  PROC DrawPart165()
    MoveL Offs(pOrigin,280.39,171.29,0.00),v40,z0,tPen\WObj:=wPaper;
    MoveL Offs(pOrigin,280.60,172.34,0.00),v40,z0,tPen\WObj:=wPaper;
    MoveL Offs(pOrigin,279.54,172.34,0.00),v40,fine,tPen\WObj:=wPaper;
    MoveL Offs(pOrigin,279.54,172.34,6.00),v60,z5,tPen\WObj:=wPaper;
    MoveL Offs(pOrigin,278.38,172.88,6.00),vTravel,z5,tPen\WObj:=wPaper;
    MoveL Offs(pOrigin,278.38,172.88,0.00),v60,z0,tPen\WObj:=wPaper;
    MoveL Offs(pOrigin,281.24,170.02,0.00),v40,fine,tPen\WObj:=wPaper;
    MoveL Offs(pOrigin,281.24,170.02,6.00),v60,z5,tPen\WObj:=wPaper;
    MoveL Offs(pOrigin,281.53,171.22,6.00),vTravel,z5,tPen\WObj:=wPaper;
    MoveL Offs(pOrigin,281.53,171.22,0.00),v60,z0,tPen\WObj:=wPaper;
    MoveL Offs(pOrigin,278.68,174.08,0.00),v40,fine,tPen\WObj:=wPaper;
    MoveL Offs(pOrigin,278.68,174.08,6.00),v60,z5,tPen\WObj:=wPaper;
    MoveL Offs(pOrigin,279.85,175.00,6.00),vTravel,z5,tPen\WObj:=wPaper;
    MoveL Offs(pOrigin,279.85,175.00,0.00),v60,z0,tPen\WObj:=wPaper;
    MoveL Offs(pOrigin,279.85,176.91,0.00),v40,z0,tPen\WObj:=wPaper;
    MoveL Offs(pOrigin,280.91,177.12,0.00),v40,z0,tPen\WObj:=wPaper;
    MoveL Offs(pOrigin,280.91,175.42,0.00),v40,z0,tPen\WObj:=wPaper;
    MoveL Offs(pOrigin,281.45,175.51,0.00),v40,z0,tPen\WObj:=wPaper;
    MoveL Offs(pOrigin,279.32,175.51,0.00),v40,z0,tPen\WObj:=wPaper;
    MoveL Offs(pOrigin,278.53,175.77,0.00),v40,z0,tPen\WObj:=wPaper;
    MoveL Offs(pOrigin,283.18,180.43,0.00),v40,z0,tPen\WObj:=wPaper;
    MoveL Offs(pOrigin,283.30,179.90,0.00),v40,z0,tPen\WObj:=wPaper;
    MoveL Offs(pOrigin,280.75,182.46,0.00),v40,z0,tPen\WObj:=wPaper;
    MoveL Offs(pOrigin,281.40,183.12,0.00),v40,z0,tPen\WObj:=wPaper;
    MoveL Offs(pOrigin,284.70,186.43,0.00),v40,z0,tPen\WObj:=wPaper;
    MoveL Offs(pOrigin,284.78,185.89,0.00),v40,z0,tPen\WObj:=wPaper;
    MoveL Offs(pOrigin,282.23,188.45,0.00),v40,z0,tPen\WObj:=wPaper;
    MoveL Offs(pOrigin,282.76,188.97,0.00),v40,z0,tPen\WObj:=wPaper;
    MoveL Offs(pOrigin,286.07,192.28,0.00),v40,z0,tPen\WObj:=wPaper;
    MoveL Offs(pOrigin,286.26,191.88,0.00),v40,z0,tPen\WObj:=wPaper;
    MoveL Offs(pOrigin,283.86,194.28,0.00),v40,z0,tPen\WObj:=wPaper;
    MoveL Offs(pOrigin,284.28,194.97,0.00),v40,z0,tPen\WObj:=wPaper;
    MoveL Offs(pOrigin,288.33,199.02,0.00),v40,z0,tPen\WObj:=wPaper;
    MoveL Offs(pOrigin,287.61,199.80,0.00),v40,z0,tPen\WObj:=wPaper;
    MoveL Offs(pOrigin,286.34,199.80,0.00),v40,z0,tPen\WObj:=wPaper;
    MoveL Offs(pOrigin,286.55,200.86,0.00),v40,z0,tPen\WObj:=wPaper;
    MoveL Offs(pOrigin,287.61,200.86,0.00),v40,z0,tPen\WObj:=wPaper;
    MoveL Offs(pOrigin,288.63,201.46,0.00),v40,z0,tPen\WObj:=wPaper;
    MoveL Offs(pOrigin,286.07,204.01,0.00),v40,z0,tPen\WObj:=wPaper;
    MoveL Offs(pOrigin,287.19,204.02,0.00),v40,z0,tPen\WObj:=wPaper;
    MoveL Offs(pOrigin,288.25,204.02,0.00),v40,z0,tPen\WObj:=wPaper;
    MoveL Offs(pOrigin,288.46,205.08,0.00),v40,z0,tPen\WObj:=wPaper;
    MoveL Offs(pOrigin,287.40,205.08,0.00),v40,fine,tPen\WObj:=wPaper;
    MoveL Offs(pOrigin,287.40,205.08,6.00),v60,z5,tPen\WObj:=wPaper;
    MoveL Offs(pOrigin,289.52,205.05,6.00),vTravel,z5,tPen\WObj:=wPaper;
    MoveL Offs(pOrigin,289.52,205.05,0.00),v60,z0,tPen\WObj:=wPaper;
    MoveL Offs(pOrigin,286.66,207.91,0.00),v40,z0,tPen\WObj:=wPaper;
    MoveL Offs(pOrigin,287.32,208.46,0.00),v40,z0,tPen\WObj:=wPaper;
    MoveL Offs(pOrigin,289.87,211.01,0.00),v40,z0,tPen\WObj:=wPaper;
    MoveL Offs(pOrigin,290.25,210.29,0.00),v40,z0,tPen\WObj:=wPaper;
    MoveL Offs(pOrigin,287.55,213.00,0.00),v40,z0,tPen\WObj:=wPaper;
    MoveL Offs(pOrigin,287.93,213.55,0.00),v40,z0,tPen\WObj:=wPaper;
    MoveL Offs(pOrigin,290.03,215.66,0.00),v40,z0,tPen\WObj:=wPaper;
    MoveL Offs(pOrigin,290.83,215.68,0.00),v40,z0,tPen\WObj:=wPaper;
    MoveL Offs(pOrigin,284.07,222.44,0.00),v40,z0,tPen\WObj:=wPaper;
    MoveL Offs(pOrigin,284.82,223.19,0.00),v40,z0,tPen\WObj:=wPaper;
    MoveL Offs(pOrigin,290.83,217.18,0.00),v40,z0,tPen\WObj:=wPaper;
    MoveL Offs(pOrigin,290.04,217.15,0.00),v40,z0,tPen\WObj:=wPaper;
    MoveL Offs(pOrigin,288.08,215.20,0.00),v40,z0,tPen\WObj:=wPaper;
    MoveL Offs(pOrigin,287.54,214.49,0.00),v40,z0,tPen\WObj:=wPaper;
    MoveL Offs(pOrigin,290.40,211.64,0.00),v40,z0,tPen\WObj:=wPaper;
    MoveL Offs(pOrigin,289.87,212.51,0.00),v40,z0,tPen\WObj:=wPaper;
    MoveL Offs(pOrigin,287.77,210.41,0.00),v40,z0,tPen\WObj:=wPaper;
    MoveL Offs(pOrigin,288.25,210.36,0.00),v40,z0,tPen\WObj:=wPaper;
    MoveL Offs(pOrigin,289.31,210.36,0.00),v40,fine,tPen\WObj:=wPaper;
    MoveL Offs(pOrigin,289.31,210.36,6.00),v60,z5,tPen\WObj:=wPaper;
    MoveL Offs(pOrigin,287.10,210.45,6.00),vTravel,z5,tPen\WObj:=wPaper;
    MoveL Offs(pOrigin,287.10,210.45,0.00),v60,z0,tPen\WObj:=wPaper;
    MoveL Offs(pOrigin,289.96,207.60,0.00),v40,fine,tPen\WObj:=wPaper;
    MoveL Offs(pOrigin,289.96,207.60,6.00),v60,z5,tPen\WObj:=wPaper;
    MoveL Offs(pOrigin,289.81,206.25,6.00),vTravel,z5,tPen\WObj:=wPaper;
    MoveL Offs(pOrigin,289.81,206.25,0.00),v60,z0,tPen\WObj:=wPaper;
    MoveL Offs(pOrigin,286.96,209.10,0.00),v40,fine,tPen\WObj:=wPaper;
    MoveL Offs(pOrigin,286.96,209.10,6.00),v60,z5,tPen\WObj:=wPaper;
    MoveL Offs(pOrigin,284.26,210.31,6.00),vTravel,z5,tPen\WObj:=wPaper;
    MoveL Offs(pOrigin,284.26,210.31,0.00),v60,z0,tPen\WObj:=wPaper;
    MoveL Offs(pOrigin,282.00,212.56,0.00),v40,z0,tPen\WObj:=wPaper;
    MoveL Offs(pOrigin,282.23,212.34,0.00),v40,z0,tPen\WObj:=wPaper;
    MoveL Offs(pOrigin,286.74,216.84,0.00),v40,fine,tPen\WObj:=wPaper;
    MoveL Offs(pOrigin,286.74,216.84,6.00),v60,z5,tPen\WObj:=wPaper;
    MoveL Offs(pOrigin,288.09,216.70,6.00),vTravel,z5,tPen\WObj:=wPaper;
    MoveL Offs(pOrigin,288.09,216.70,0.00),v60,z0,tPen\WObj:=wPaper;
    MoveL Offs(pOrigin,290.04,218.65,0.00),v40,z0,tPen\WObj:=wPaper;
    MoveL Offs(pOrigin,290.52,218.98,0.00),v40,z0,tPen\WObj:=wPaper;
    MoveL Offs(pOrigin,285.26,224.24,0.00),v40,z0,tPen\WObj:=wPaper;
    MoveL Offs(pOrigin,285.86,225.13,0.00),v40,z0,tPen\WObj:=wPaper;
    MoveL Offs(pOrigin,290.82,220.18,0.00),v40,z0,tPen\WObj:=wPaper;
    MoveL Offs(pOrigin,291.85,220.46,0.00),v40,z0,tPen\WObj:=wPaper;
    MoveL Offs(pOrigin,293.35,221.96,0.00),v40,z0,tPen\WObj:=wPaper;
    MoveL Offs(pOrigin,292.71,222.18,0.00),v40,z0,tPen\WObj:=wPaper;
    MoveL Offs(pOrigin,292.50,222.60,0.00),v40,z0,tPen\WObj:=wPaper;
    MoveL Offs(pOrigin,292.71,222.18,0.00),v40,z0,tPen\WObj:=wPaper;
    MoveL Offs(pOrigin,292.50,221.98,0.00),v40,z0,tPen\WObj:=wPaper;
    MoveL Offs(pOrigin,291.23,221.98,0.00),v40,z0,tPen\WObj:=wPaper;
    MoveL Offs(pOrigin,291.25,221.35,0.00),v40,z0,tPen\WObj:=wPaper;
    MoveL Offs(pOrigin,292.60,222.70,0.00),v40,z0,tPen\WObj:=wPaper;
    MoveL Offs(pOrigin,292.08,222.81,0.00),v40,z0,tPen\WObj:=wPaper;
    MoveL Offs(pOrigin,291.86,223.24,0.00),v40,z0,tPen\WObj:=wPaper;
    MoveL Offs(pOrigin,292.08,222.81,0.00),v40,z0,tPen\WObj:=wPaper;
    MoveL Offs(pOrigin,291.65,223.03,0.00),v40,z0,tPen\WObj:=wPaper;
    MoveL Offs(pOrigin,286.12,223.03,0.00),v40,z0,tPen\WObj:=wPaper;
    MoveL Offs(pOrigin,286.55,222.39,0.00),v40,z0,tPen\WObj:=wPaper;
    MoveL Offs(pOrigin,286.98,223.66,0.00),v40,z0,tPen\WObj:=wPaper;
    MoveL Offs(pOrigin,286.55,223.88,0.00),v40,z0,tPen\WObj:=wPaper;
    MoveL Offs(pOrigin,286.55,223.88,0.00),v40,z0,tPen\WObj:=wPaper;
    MoveL Offs(pOrigin,285.91,223.45,0.00),v40,z0,tPen\WObj:=wPaper;
    MoveL Offs(pOrigin,283.43,219.62,0.00),v40,z0,tPen\WObj:=wPaper;
    MoveL Offs(pOrigin,283.79,219.48,0.00),v40,z0,tPen\WObj:=wPaper;
    MoveL Offs(pOrigin,284.42,219.84,0.00),v40,z0,tPen\WObj:=wPaper;
    MoveL Offs(pOrigin,285.91,221.96,0.00),v40,z0,tPen\WObj:=wPaper;
    MoveL Offs(pOrigin,286.55,222.39,0.00),v40,z0,tPen\WObj:=wPaper;
    MoveL Offs(pOrigin,286.55,222.39,0.00),v40,z0,tPen\WObj:=wPaper;
    MoveL Offs(pOrigin,286.76,221.54,0.00),v40,z0,tPen\WObj:=wPaper;
    MoveL Offs(pOrigin,284.71,216.01,0.00),v40,z0,tPen\WObj:=wPaper;
    MoveL Offs(pOrigin,282.65,211.76,0.00),v40,z0,tPen\WObj:=wPaper;
    MoveL Offs(pOrigin,279.47,207.30,0.00),v40,z0,tPen\WObj:=wPaper;
    MoveL Offs(pOrigin,278.69,205.39,0.00),v40,z0,tPen\WObj:=wPaper;
    MoveL Offs(pOrigin,272.10,200.64,0.00),v40,z0,tPen\WObj:=wPaper;
    MoveL Offs(pOrigin,267.64,198.38,0.00),v40,fine,tPen\WObj:=wPaper;
    MoveL Offs(pOrigin,267.64,198.38,6.00),v60,z5,tPen\WObj:=wPaper;
  ENDPROC

  PROC DrawPart166()
    MoveL Offs(pOrigin,269.31,199.87,6.00),vTravel,z5,tPen\WObj:=wPaper;
    MoveL Offs(pOrigin,269.31,199.87,0.00),v60,z0,tPen\WObj:=wPaper;
    MoveL Offs(pOrigin,270.51,198.67,0.00),v40,z0,tPen\WObj:=wPaper;
    MoveL Offs(pOrigin,271.56,199.11,0.00),v40,z0,tPen\WObj:=wPaper;
    MoveL Offs(pOrigin,270.21,200.47,0.00),v40,z0,tPen\WObj:=wPaper;
    MoveL Offs(pOrigin,271.10,201.06,0.00),v40,z0,tPen\WObj:=wPaper;
    MoveL Offs(pOrigin,272.46,199.71,0.00),v40,z0,tPen\WObj:=wPaper;
    MoveL Offs(pOrigin,271.86,200.47,0.00),v40,z0,tPen\WObj:=wPaper;
    MoveL Offs(pOrigin,275.62,204.23,0.00),v40,z0,tPen\WObj:=wPaper;
    MoveL Offs(pOrigin,275.14,204.50,0.00),v40,z0,tPen\WObj:=wPaper;
    MoveL Offs(pOrigin,279.04,200.59,0.00),v40,z0,tPen\WObj:=wPaper;
    MoveL Offs(pOrigin,278.26,200.86,0.00),v40,z0,tPen\WObj:=wPaper;
    MoveL Offs(pOrigin,276.99,200.86,0.00),v40,fine,tPen\WObj:=wPaper;
    MoveL Offs(pOrigin,276.99,200.86,6.00),v60,z5,tPen\WObj:=wPaper;
    MoveL Offs(pOrigin,277.62,201.91,6.00),vTravel,z5,tPen\WObj:=wPaper;
    MoveL Offs(pOrigin,277.62,201.91,0.00),v60,z0,tPen\WObj:=wPaper;
    MoveL Offs(pOrigin,278.90,201.91,0.00),v40,z0,tPen\WObj:=wPaper;
    MoveL Offs(pOrigin,279.11,201.99,0.00),v40,z0,tPen\WObj:=wPaper;
    MoveL Offs(pOrigin,279.54,202.62,0.00),v40,z0,tPen\WObj:=wPaper;
    MoveL Offs(pOrigin,279.11,201.99,0.00),v40,z0,tPen\WObj:=wPaper;
    MoveL Offs(pOrigin,279.51,202.14,0.00),v40,z0,tPen\WObj:=wPaper;
    MoveL Offs(pOrigin,271.69,194.33,0.00),v40,fine,tPen\WObj:=wPaper;
    MoveL Offs(pOrigin,271.69,194.33,6.00),v60,z5,tPen\WObj:=wPaper;
    MoveL Offs(pOrigin,272.52,193.46,6.00),vTravel,z5,tPen\WObj:=wPaper;
    MoveL Offs(pOrigin,272.52,193.46,0.00),v60,z0,tPen\WObj:=wPaper;
    MoveL Offs(pOrigin,273.80,193.46,0.00),v40,z0,tPen\WObj:=wPaper;
    MoveL Offs(pOrigin,274.01,193.49,0.00),v40,z0,tPen\WObj:=wPaper;
    MoveL Offs(pOrigin,274.44,194.12,0.00),v40,z0,tPen\WObj:=wPaper;
    MoveL Offs(pOrigin,274.01,193.49,0.00),v40,z0,tPen\WObj:=wPaper;
    MoveL Offs(pOrigin,274.57,193.11,0.00),v40,z0,tPen\WObj:=wPaper;
    MoveL Offs(pOrigin,271.12,196.57,0.00),v40,z0,tPen\WObj:=wPaper;
    MoveL Offs(pOrigin,271.86,197.32,0.00),v40,z0,tPen\WObj:=wPaper;
    MoveL Offs(pOrigin,275.17,194.01,0.00),v40,z0,tPen\WObj:=wPaper;
    MoveL Offs(pOrigin,275.14,194.79,0.00),v40,z0,tPen\WObj:=wPaper;
    MoveL Offs(pOrigin,266.42,186.07,0.00),v40,z0,tPen\WObj:=wPaper;
    MoveL Offs(pOrigin,266.79,185.20,0.00),v40,z0,tPen\WObj:=wPaper;
    MoveL Offs(pOrigin,267.00,185.62,0.00),v40,z0,tPen\WObj:=wPaper;
    MoveL Offs(pOrigin,266.79,185.20,0.00),v40,z0,tPen\WObj:=wPaper;
    MoveL Offs(pOrigin,267.00,185.02,0.00),v40,z0,tPen\WObj:=wPaper;
    MoveL Offs(pOrigin,268.27,185.02,0.00),v40,z0,tPen\WObj:=wPaper;
    MoveL Offs(pOrigin,268.49,185.20,0.00),v40,z0,tPen\WObj:=wPaper;
    MoveL Offs(pOrigin,268.70,185.62,0.00),v40,z0,tPen\WObj:=wPaper;
    MoveL Offs(pOrigin,268.49,185.20,0.00),v40,z0,tPen\WObj:=wPaper;
    MoveL Offs(pOrigin,269.12,186.07,0.00),v40,z0,tPen\WObj:=wPaper;
    MoveL Offs(pOrigin,267.64,186.07,0.00),v40,z0,tPen\WObj:=wPaper;
    MoveL Offs(pOrigin,267.85,187.13,0.00),v40,z0,tPen\WObj:=wPaper;
    MoveL Offs(pOrigin,269.76,187.13,0.00),v40,z0,tPen\WObj:=wPaper;
    MoveL Offs(pOrigin,269.76,187.11,0.00),v40,z0,tPen\WObj:=wPaper;
    MoveL Offs(pOrigin,270.19,187.75,0.00),v40,z0,tPen\WObj:=wPaper;
    MoveL Offs(pOrigin,269.76,187.11,0.00),v40,z0,tPen\WObj:=wPaper;
    MoveL Offs(pOrigin,269.29,187.96,0.00),v40,z0,tPen\WObj:=wPaper;
    MoveL Offs(pOrigin,269.29,189.02,0.00),v40,z0,tPen\WObj:=wPaper;
    MoveL Offs(pOrigin,269.12,189.24,0.00),v40,z0,tPen\WObj:=wPaper;
    MoveL Offs(pOrigin,271.25,189.24,0.00),v40,z0,tPen\WObj:=wPaper;
    MoveL Offs(pOrigin,270.35,189.02,0.00),v40,z0,tPen\WObj:=wPaper;
    MoveL Offs(pOrigin,270.35,190.09,0.00),v40,z0,tPen\WObj:=wPaper;
    MoveL Offs(pOrigin,269.98,190.30,0.00),v40,z0,tPen\WObj:=wPaper;
    MoveL Offs(pOrigin,271.68,190.30,0.00),v40,fine,tPen\WObj:=wPaper;
    MoveL Offs(pOrigin,271.68,190.30,6.00),v60,z5,tPen\WObj:=wPaper;
    MoveL Offs(pOrigin,272.58,189.24,6.00),vTravel,z5,tPen\WObj:=wPaper;
    MoveL Offs(pOrigin,272.58,189.24,0.00),v60,z0,tPen\WObj:=wPaper;
    MoveL Offs(pOrigin,260.10,176.77,0.00),v40,z0,tPen\WObj:=wPaper;
    MoveL Offs(pOrigin,259.34,176.98,0.00),v40,z0,tPen\WObj:=wPaper;
    MoveL Offs(pOrigin,262.20,174.13,0.00),v40,z0,tPen\WObj:=wPaper;
    MoveL Offs(pOrigin,261.44,173.62,0.00),v40,z0,tPen\WObj:=wPaper;
    MoveL Offs(pOrigin,258.14,170.32,0.00),v40,z0,tPen\WObj:=wPaper;
    MoveL Offs(pOrigin,258.01,170.84,0.00),v40,z0,tPen\WObj:=wPaper;
    MoveL Offs(pOrigin,260.42,168.44,0.00),v40,z0,tPen\WObj:=wPaper;
    MoveL Offs(pOrigin,259.67,167.69,0.00),v40,z0,tPen\WObj:=wPaper;
    MoveL Offs(pOrigin,257.57,169.80,0.00),v40,z0,tPen\WObj:=wPaper;
    MoveL Offs(pOrigin,256.82,169.05,0.00),v40,z0,tPen\WObj:=wPaper;
    MoveL Offs(pOrigin,259.08,166.80,0.00),v40,z0,tPen\WObj:=wPaper;
    MoveL Offs(pOrigin,258.48,165.90,0.00),v40,z0,tPen\WObj:=wPaper;
    MoveL Offs(pOrigin,256.07,168.30,0.00),v40,z0,tPen\WObj:=wPaper;
    MoveL Offs(pOrigin,255.33,167.56,0.00),v40,z0,tPen\WObj:=wPaper;
    MoveL Offs(pOrigin,257.58,165.30,0.00),v40,z0,tPen\WObj:=wPaper;
    MoveL Offs(pOrigin,256.80,166.01,0.00),v40,z0,tPen\WObj:=wPaper;
    MoveL Offs(pOrigin,255.31,166.01,0.00),v40,z0,tPen\WObj:=wPaper;
    MoveL Offs(pOrigin,255.74,166.71,0.00),v40,z0,tPen\WObj:=wPaper;
    MoveL Offs(pOrigin,257.86,168.84,0.00),v40,z0,tPen\WObj:=wPaper;
    MoveL Offs(pOrigin,255.74,166.71,0.00),v40,z0,tPen\WObj:=wPaper;
    MoveL Offs(pOrigin,256.38,167.06,0.00),v40,z0,tPen\WObj:=wPaper;
    MoveL Offs(pOrigin,257.86,167.06,0.00),v40,z0,tPen\WObj:=wPaper;
    MoveL Offs(pOrigin,257.44,168.12,0.00),v40,z0,tPen\WObj:=wPaper;
    MoveL Offs(pOrigin,258.92,168.12,0.00),v40,z0,tPen\WObj:=wPaper;
    MoveL Offs(pOrigin,258.92,167.99,0.00),v40,z0,tPen\WObj:=wPaper;
    MoveL Offs(pOrigin,259.35,168.41,0.00),v40,z0,tPen\WObj:=wPaper;
    MoveL Offs(pOrigin,258.92,167.99,0.00),v40,fine,tPen\WObj:=wPaper;
    MoveL Offs(pOrigin,258.92,167.99,6.00),v60,z5,tPen\WObj:=wPaper;
    MoveL Offs(pOrigin,258.50,169.18,6.00),vTravel,z5,tPen\WObj:=wPaper;
    MoveL Offs(pOrigin,258.50,169.18,0.00),v60,z0,tPen\WObj:=wPaper;
    MoveL Offs(pOrigin,259.56,169.18,0.00),v40,z0,tPen\WObj:=wPaper;
    MoveL Offs(pOrigin,260.38,169.58,0.00),v40,z0,tPen\WObj:=wPaper;
    MoveL Offs(pOrigin,246.26,155.45,0.00),v40,z0,tPen\WObj:=wPaper;
    MoveL Offs(pOrigin,245.93,156.05,0.00),v40,z0,tPen\WObj:=wPaper;
    MoveL Offs(pOrigin,248.03,153.95,0.00),v40,fine,tPen\WObj:=wPaper;
    MoveL Offs(pOrigin,248.03,153.95,6.00),v60,z5,tPen\WObj:=wPaper;
    MoveL Offs(pOrigin,247.73,152.75,6.00),vTravel,z5,tPen\WObj:=wPaper;
    MoveL Offs(pOrigin,247.73,152.75,0.00),v60,z0,tPen\WObj:=wPaper;
    MoveL Offs(pOrigin,245.63,154.85,0.00),v40,fine,tPen\WObj:=wPaper;
    MoveL Offs(pOrigin,245.63,154.85,6.00),v60,z5,tPen\WObj:=wPaper;
    MoveL Offs(pOrigin,245.33,153.66,6.00),vTravel,z5,tPen\WObj:=wPaper;
    MoveL Offs(pOrigin,245.33,153.66,0.00),v60,z0,tPen\WObj:=wPaper;
    MoveL Offs(pOrigin,247.44,151.55,0.00),v40,z0,tPen\WObj:=wPaper;
    MoveL Offs(pOrigin,246.99,150.50,0.00),v40,z0,tPen\WObj:=wPaper;
    MoveL Offs(pOrigin,245.04,152.46,0.00),v40,fine,tPen\WObj:=wPaper;
    MoveL Offs(pOrigin,245.04,152.46,6.00),v60,z5,tPen\WObj:=wPaper;
    MoveL Offs(pOrigin,244.74,151.26,6.00),vTravel,z5,tPen\WObj:=wPaper;
    MoveL Offs(pOrigin,244.74,151.26,0.00),v60,z0,tPen\WObj:=wPaper;
    MoveL Offs(pOrigin,246.70,149.31,0.00),v40,z0,tPen\WObj:=wPaper;
    MoveL Offs(pOrigin,246.39,149.61,0.00),v40,z0,tPen\WObj:=wPaper;
    MoveL Offs(pOrigin,244.89,148.11,0.00),v40,z0,tPen\WObj:=wPaper;
    MoveL Offs(pOrigin,244.30,148.72,0.00),v40,z0,tPen\WObj:=wPaper;
    MoveL Offs(pOrigin,246.55,146.46,0.00),v40,fine,tPen\WObj:=wPaper;
    MoveL Offs(pOrigin,246.55,146.46,6.00),v60,z5,tPen\WObj:=wPaper;
    MoveL Offs(pOrigin,246.26,145.26,6.00),vTravel,z5,tPen\WObj:=wPaper;
    MoveL Offs(pOrigin,246.26,145.26,0.00),v60,z0,tPen\WObj:=wPaper;
    MoveL Offs(pOrigin,244.16,147.37,0.00),v40,fine,tPen\WObj:=wPaper;
    MoveL Offs(pOrigin,244.16,147.37,6.00),v60,z5,tPen\WObj:=wPaper;
    MoveL Offs(pOrigin,245.11,144.82,6.00),vTravel,z5,tPen\WObj:=wPaper;
  ENDPROC

  PROC DrawPart167()
    MoveL Offs(pOrigin,245.11,144.82,0.00),v60,z0,tPen\WObj:=wPaper;
    MoveL Offs(pOrigin,244.69,144.40,0.00),v40,z0,tPen\WObj:=wPaper;
    MoveL Offs(pOrigin,244.90,143.34,0.00),v40,z0,tPen\WObj:=wPaper;
    MoveL Offs(pOrigin,244.90,142.27,0.00),v40,z0,tPen\WObj:=wPaper;
    MoveL Offs(pOrigin,244.48,141.85,0.00),v40,z0,tPen\WObj:=wPaper;
    MoveL Offs(pOrigin,244.69,140.79,0.00),v40,fine,tPen\WObj:=wPaper;
    MoveL Offs(pOrigin,244.69,140.79,6.00),v60,z5,tPen\WObj:=wPaper;
    MoveL Offs(pOrigin,239.98,141.09,6.00),vTravel,z5,tPen\WObj:=wPaper;
    MoveL Offs(pOrigin,239.98,141.09,0.00),v60,z0,tPen\WObj:=wPaper;
    MoveL Offs(pOrigin,238.33,142.74,0.00),v40,z0,tPen\WObj:=wPaper;
    MoveL Offs(pOrigin,239.22,143.34,0.00),v40,z0,tPen\WObj:=wPaper;
    MoveL Offs(pOrigin,237.12,145.44,0.00),v40,fine,tPen\WObj:=wPaper;
    MoveL Offs(pOrigin,237.12,145.44,6.00),v60,z5,tPen\WObj:=wPaper;
    MoveL Offs(pOrigin,238.62,145.44,6.00),vTravel,z5,tPen\WObj:=wPaper;
    MoveL Offs(pOrigin,238.62,145.44,0.00),v60,z0,tPen\WObj:=wPaper;
    MoveL Offs(pOrigin,235.61,148.44,0.00),v40,fine,tPen\WObj:=wPaper;
    MoveL Offs(pOrigin,235.61,148.44,6.00),v60,z5,tPen\WObj:=wPaper;
    MoveL Offs(pOrigin,237.11,149.94,6.00),vTravel,z5,tPen\WObj:=wPaper;
    MoveL Offs(pOrigin,237.11,149.94,0.00),v60,z0,tPen\WObj:=wPaper;
    MoveL Offs(pOrigin,233.20,153.84,0.00),v40,fine,tPen\WObj:=wPaper;
    MoveL Offs(pOrigin,233.20,153.84,6.00),v60,z5,tPen\WObj:=wPaper;
    MoveL Offs(pOrigin,235.29,154.73,6.00),vTravel,z5,tPen\WObj:=wPaper;
    MoveL Offs(pOrigin,235.29,154.73,0.00),v60,z0,tPen\WObj:=wPaper;
    MoveL Offs(pOrigin,226.43,163.60,0.00),v40,z0,tPen\WObj:=wPaper;
    MoveL Offs(pOrigin,227.11,163.18,0.00),v40,z0,tPen\WObj:=wPaper;
    MoveL Offs(pOrigin,230.26,166.34,0.00),v40,z0,tPen\WObj:=wPaper;
    MoveL Offs(pOrigin,230.91,166.58,0.00),v40,z0,tPen\WObj:=wPaper;
    MoveL Offs(pOrigin,225.50,171.99,0.00),v40,fine,tPen\WObj:=wPaper;
    MoveL Offs(pOrigin,225.50,171.99,6.00),v60,z5,tPen\WObj:=wPaper;
    MoveL Offs(pOrigin,225.35,173.64,6.00),vTravel,z5,tPen\WObj:=wPaper;
    MoveL Offs(pOrigin,225.35,173.64,0.00),v60,z0,tPen\WObj:=wPaper;
    MoveL Offs(pOrigin,230.01,168.98,0.00),v40,z0,tPen\WObj:=wPaper;
    MoveL Offs(pOrigin,229.52,168.58,0.00),v40,z0,tPen\WObj:=wPaper;
    MoveL Offs(pOrigin,226.82,165.88,0.00),v40,z0,tPen\WObj:=wPaper;
    MoveL Offs(pOrigin,227.26,166.01,0.00),v40,z0,tPen\WObj:=wPaper;
    MoveL Offs(pOrigin,229.60,166.01,0.00),v40,z0,tPen\WObj:=wPaper;
    MoveL Offs(pOrigin,229.39,167.06,0.00),v40,z0,tPen\WObj:=wPaper;
    MoveL Offs(pOrigin,227.26,167.06,0.00),v40,z0,tPen\WObj:=wPaper;
    MoveL Offs(pOrigin,227.05,168.12,0.00),v40,z0,tPen\WObj:=wPaper;
    MoveL Offs(pOrigin,229.18,168.12,0.00),v40,fine,tPen\WObj:=wPaper;
    MoveL Offs(pOrigin,229.18,168.12,6.00),v60,z5,tPen\WObj:=wPaper;
    MoveL Offs(pOrigin,228.54,170.23,6.00),vTravel,z5,tPen\WObj:=wPaper;
    MoveL Offs(pOrigin,228.54,170.23,0.00),v60,z0,tPen\WObj:=wPaper;
    MoveL Offs(pOrigin,226.84,170.23,0.00),v40,z0,tPen\WObj:=wPaper;
    MoveL Offs(pOrigin,227.05,169.48,0.00),v40,z0,tPen\WObj:=wPaper;
    MoveL Offs(pOrigin,227.05,175.21,0.00),v40,z0,tPen\WObj:=wPaper;
    MoveL Offs(pOrigin,228.11,174.79,0.00),v40,z0,tPen\WObj:=wPaper;
    MoveL Offs(pOrigin,228.11,165.22,0.00),v40,fine,tPen\WObj:=wPaper;
    MoveL Offs(pOrigin,228.11,165.22,6.00),v60,z5,tPen\WObj:=wPaper;
    MoveL Offs(pOrigin,227.69,163.90,6.00),vTravel,z5,tPen\WObj:=wPaper;
    MoveL Offs(pOrigin,227.69,163.90,0.00),v60,z0,tPen\WObj:=wPaper;
    MoveL Offs(pOrigin,229.39,163.90,0.00),v40,z0,tPen\WObj:=wPaper;
    MoveL Offs(pOrigin,229.18,162.84,0.00),v40,z0,tPen\WObj:=wPaper;
    MoveL Offs(pOrigin,227.90,162.84,0.00),v40,z0,tPen\WObj:=wPaper;
    MoveL Offs(pOrigin,227.40,161.99,0.00),v40,z0,tPen\WObj:=wPaper;
    MoveL Offs(pOrigin,230.71,165.29,0.00),v40,z0,tPen\WObj:=wPaper;
    MoveL Offs(pOrigin,231.37,164.63,0.00),v40,z0,tPen\WObj:=wPaper;
    MoveL Offs(pOrigin,225.66,170.34,0.00),v40,fine,tPen\WObj:=wPaper;
    MoveL Offs(pOrigin,225.66,170.34,6.00),v60,z5,tPen\WObj:=wPaper;
    MoveL Offs(pOrigin,229.40,171.08,6.00),vTravel,z5,tPen\WObj:=wPaper;
    MoveL Offs(pOrigin,229.40,171.08,0.00),v60,z0,tPen\WObj:=wPaper;
    MoveL Offs(pOrigin,225.04,175.44,0.00),v40,fine,tPen\WObj:=wPaper;
    MoveL Offs(pOrigin,225.04,175.44,6.00),v60,z5,tPen\WObj:=wPaper;
    MoveL Offs(pOrigin,225.99,176.57,6.00),vTravel,z5,tPen\WObj:=wPaper;
    MoveL Offs(pOrigin,225.99,176.57,0.00),v60,z0,tPen\WObj:=wPaper;
    MoveL Offs(pOrigin,229.39,176.57,0.00),v40,z0,tPen\WObj:=wPaper;
    MoveL Offs(pOrigin,229.60,177.62,0.00),v40,z0,tPen\WObj:=wPaper;
    MoveL Offs(pOrigin,228.32,177.62,0.00),v40,z0,tPen\WObj:=wPaper;
    MoveL Offs(pOrigin,227.26,177.62,0.00),v40,z0,tPen\WObj:=wPaper;
    MoveL Offs(pOrigin,225.78,177.62,0.00),v40,z0,tPen\WObj:=wPaper;
    MoveL Offs(pOrigin,225.35,177.86,0.00),v40,z0,tPen\WObj:=wPaper;
    MoveL Offs(pOrigin,230.31,182.82,0.00),v40,z0,tPen\WObj:=wPaper;
    MoveL Offs(pOrigin,230.86,183.06,0.00),v40,z0,tPen\WObj:=wPaper;
    MoveL Offs(pOrigin,228.31,185.61,0.00),v40,z0,tPen\WObj:=wPaper;
    MoveL Offs(pOrigin,228.52,185.51,0.00),v40,z0,tPen\WObj:=wPaper;
    MoveL Offs(pOrigin,231.83,188.81,0.00),v40,z0,tPen\WObj:=wPaper;
    MoveL Offs(pOrigin,231.00,188.90,0.00),v40,z0,tPen\WObj:=wPaper;
    MoveL Offs(pOrigin,245.12,174.78,0.00),v40,z0,tPen\WObj:=wPaper;
    MoveL Offs(pOrigin,244.67,174.77,0.00),v40,z0,tPen\WObj:=wPaper;
    MoveL Offs(pOrigin,243.17,173.27,0.00),v40,z0,tPen\WObj:=wPaper;
    MoveL Offs(pOrigin,242.43,172.99,0.00),v40,z0,tPen\WObj:=wPaper;
    MoveL Offs(pOrigin,253.70,161.72,0.00),v40,z0,tPen\WObj:=wPaper;
    MoveL Offs(pOrigin,252.95,160.97,0.00),v40,z0,tPen\WObj:=wPaper;
    MoveL Offs(pOrigin,250.55,163.38,0.00),v40,z0,tPen\WObj:=wPaper;
    MoveL Offs(pOrigin,250.92,163.11,0.00),v40,z0,tPen\WObj:=wPaper;
    MoveL Offs(pOrigin,253.63,165.81,0.00),v40,z0,tPen\WObj:=wPaper;
    MoveL Offs(pOrigin,253.68,166.21,0.00),v40,z0,tPen\WObj:=wPaper;
    MoveL Offs(pOrigin,256.09,163.81,0.00),v40,z0,tPen\WObj:=wPaper;
    MoveL Offs(pOrigin,256.84,163.06,0.00),v40,z0,tPen\WObj:=wPaper;
    MoveL Offs(pOrigin,257.59,162.31,0.00),v40,z0,tPen\WObj:=wPaper;
    MoveL Offs(pOrigin,258.64,162.75,0.00),v40,z0,tPen\WObj:=wPaper;
    MoveL Offs(pOrigin,257.59,163.80,0.00),v40,z0,tPen\WObj:=wPaper;
    MoveL Offs(pOrigin,258.33,164.55,0.00),v40,z0,tPen\WObj:=wPaper;
    MoveL Offs(pOrigin,259.54,163.35,0.00),v40,z0,tPen\WObj:=wPaper;
    MoveL Offs(pOrigin,260.58,163.79,0.00),v40,z0,tPen\WObj:=wPaper;
    MoveL Offs(pOrigin,259.23,165.15,0.00),v40,z0,tPen\WObj:=wPaper;
    MoveL Offs(pOrigin,260.13,165.74,0.00),v40,z0,tPen\WObj:=wPaper;
    MoveL Offs(pOrigin,261.78,164.09,0.00),v40,z0,tPen\WObj:=wPaper;
    MoveL Offs(pOrigin,262.53,164.84,0.00),v40,z0,tPen\WObj:=wPaper;
    MoveL Offs(pOrigin,260.72,166.64,0.00),v40,z0,tPen\WObj:=wPaper;
    MoveL Offs(pOrigin,261.42,166.13,0.00),v40,z0,tPen\WObj:=wPaper;
    MoveL Offs(pOrigin,265.93,170.64,0.00),v40,z0,tPen\WObj:=wPaper;
    MoveL Offs(pOrigin,265.20,171.12,0.00),v40,z0,tPen\WObj:=wPaper;
    MoveL Offs(pOrigin,266.56,169.77,0.00),v40,z0,tPen\WObj:=wPaper;
    MoveL Offs(pOrigin,265.81,169.02,0.00),v40,z0,tPen\WObj:=wPaper;
    MoveL Offs(pOrigin,264.31,170.52,0.00),v40,z0,tPen\WObj:=wPaper;
    MoveL Offs(pOrigin,263.71,169.63,0.00),v40,z0,tPen\WObj:=wPaper;
    MoveL Offs(pOrigin,265.21,168.12,0.00),v40,z0,tPen\WObj:=wPaper;
    MoveL Offs(pOrigin,264.47,167.38,0.00),v40,z0,tPen\WObj:=wPaper;
    MoveL Offs(pOrigin,262.96,168.88,0.00),v40,z0,tPen\WObj:=wPaper;
    MoveL Offs(pOrigin,262.22,168.13,0.00),v40,z0,tPen\WObj:=wPaper;
    MoveL Offs(pOrigin,263.72,166.63,0.00),v40,z0,tPen\WObj:=wPaper;
    MoveL Offs(pOrigin,263.12,165.73,0.00),v40,z0,tPen\WObj:=wPaper;
    MoveL Offs(pOrigin,261.32,167.54,0.00),v40,fine,tPen\WObj:=wPaper;
    MoveL Offs(pOrigin,261.32,167.54,6.00),v60,z5,tPen\WObj:=wPaper;
    MoveL Offs(pOrigin,262.33,166.07,6.00),vTravel,z5,tPen\WObj:=wPaper;
    MoveL Offs(pOrigin,262.33,166.07,0.00),v60,z0,tPen\WObj:=wPaper;
    MoveL Offs(pOrigin,261.05,159.06,0.00),v40,z0,tPen\WObj:=wPaper;
    MoveL Offs(pOrigin,260.41,150.56,0.00),v40,z0,tPen\WObj:=wPaper;
    MoveL Offs(pOrigin,259.35,110.82,0.00),v40,z0,tPen\WObj:=wPaper;
  ENDPROC

  PROC DrawPart168()
    MoveL Offs(pOrigin,258.50,94.46,0.00),v40,z0,tPen\WObj:=wPaper;
    MoveL Offs(pOrigin,258.92,94.04,0.00),v40,z0,tPen\WObj:=wPaper;
    MoveL Offs(pOrigin,259.55,94.08,0.00),v40,z0,tPen\WObj:=wPaper;
    MoveL Offs(pOrigin,258.65,93.17,0.00),v40,z0,tPen\WObj:=wPaper;
    MoveL Offs(pOrigin,257.80,93.40,0.00),v40,z0,tPen\WObj:=wPaper;
    MoveL Offs(pOrigin,259.31,91.90,0.00),v40,z0,tPen\WObj:=wPaper;
    MoveL Offs(pOrigin,260.05,92.64,0.00),v40,z0,tPen\WObj:=wPaper;
    MoveL Offs(pOrigin,258.10,94.60,0.00),v40,fine,tPen\WObj:=wPaper;
    MoveL Offs(pOrigin,258.10,94.60,6.00),v60,z5,tPen\WObj:=wPaper;
    MoveL Offs(pOrigin,258.39,95.79,6.00),vTravel,z5,tPen\WObj:=wPaper;
    MoveL Offs(pOrigin,258.39,95.79,0.00),v60,z0,tPen\WObj:=wPaper;
    MoveL Offs(pOrigin,260.50,93.69,0.00),v40,z0,tPen\WObj:=wPaper;
    MoveL Offs(pOrigin,261.09,94.59,0.00),v40,z0,tPen\WObj:=wPaper;
    MoveL Offs(pOrigin,259.14,96.54,0.00),v40,z0,tPen\WObj:=wPaper;
    MoveL Offs(pOrigin,259.74,97.44,0.00),v40,z0,tPen\WObj:=wPaper;
    MoveL Offs(pOrigin,261.54,95.63,0.00),v40,z0,tPen\WObj:=wPaper;
    MoveL Offs(pOrigin,261.99,96.68,0.00),v40,z0,tPen\WObj:=wPaper;
    MoveL Offs(pOrigin,260.33,98.33,0.00),v40,z0,tPen\WObj:=wPaper;
    MoveL Offs(pOrigin,260.93,99.23,0.00),v40,z0,tPen\WObj:=wPaper;
    MoveL Offs(pOrigin,262.58,97.58,0.00),v40,z0,tPen\WObj:=wPaper;
    MoveL Offs(pOrigin,261.48,97.65,0.00),v40,z0,tPen\WObj:=wPaper;
    MoveL Offs(pOrigin,261.69,98.07,0.00),v40,z0,tPen\WObj:=wPaper;
    MoveL Offs(pOrigin,261.48,97.65,0.00),v40,z0,tPen\WObj:=wPaper;
    MoveL Offs(pOrigin,261.05,96.80,0.00),v40,z0,tPen\WObj:=wPaper;
    MoveL Offs(pOrigin,261.26,97.22,0.00),v40,z0,tPen\WObj:=wPaper;
    MoveL Offs(pOrigin,261.05,96.80,0.00),v40,fine,tPen\WObj:=wPaper;
    MoveL Offs(pOrigin,261.05,96.80,6.00),v60,z5,tPen\WObj:=wPaper;
    MoveL Offs(pOrigin,260.20,95.10,6.00),vTravel,z5,tPen\WObj:=wPaper;
    MoveL Offs(pOrigin,260.20,95.10,0.00),v60,z0,tPen\WObj:=wPaper;
    MoveL Offs(pOrigin,260.41,95.53,0.00),v40,z0,tPen\WObj:=wPaper;
    MoveL Offs(pOrigin,260.20,95.10,0.00),v40,fine,tPen\WObj:=wPaper;
    MoveL Offs(pOrigin,260.20,95.10,6.00),v60,z5,tPen\WObj:=wPaper;
    MoveL Offs(pOrigin,257.36,92.35,6.00),vTravel,z5,tPen\WObj:=wPaper;
    MoveL Offs(pOrigin,257.36,92.35,0.00),v60,z0,tPen\WObj:=wPaper;
    MoveL Offs(pOrigin,259.01,90.70,0.00),v40,z0,tPen\WObj:=wPaper;
    MoveL Offs(pOrigin,258.56,89.65,0.00),v40,z0,tPen\WObj:=wPaper;
    MoveL Offs(pOrigin,256.91,91.30,0.00),v40,z0,tPen\WObj:=wPaper;
    MoveL Offs(pOrigin,256.46,90.26,0.00),v40,z0,tPen\WObj:=wPaper;
    MoveL Offs(pOrigin,258.12,88.60,0.00),v40,z0,tPen\WObj:=wPaper;
    MoveL Offs(pOrigin,257.67,87.56,0.00),v40,z0,tPen\WObj:=wPaper;
    MoveL Offs(pOrigin,256.02,89.21,0.00),v40,z0,tPen\WObj:=wPaper;
    MoveL Offs(pOrigin,255.57,88.16,0.00),v40,z0,tPen\WObj:=wPaper;
    MoveL Offs(pOrigin,256.62,87.11,0.00),v40,z0,tPen\WObj:=wPaper;
    MoveL Offs(pOrigin,255.88,86.36,0.00),v40,z0,tPen\WObj:=wPaper;
    MoveL Offs(pOrigin,254.98,87.26,0.00),v40,z0,tPen\WObj:=wPaper;
    MoveL Offs(pOrigin,254.53,86.22,0.00),v40,z0,tPen\WObj:=wPaper;
    MoveL Offs(pOrigin,255.28,85.47,0.00),v40,fine,tPen\WObj:=wPaper;
    MoveL Offs(pOrigin,255.28,85.47,6.00),v60,z5,tPen\WObj:=wPaper;
    MoveL Offs(pOrigin,257.23,89.57,6.00),vTravel,z5,tPen\WObj:=wPaper;
    MoveL Offs(pOrigin,257.23,89.57,0.00),v60,z0,tPen\WObj:=wPaper;
    MoveL Offs(pOrigin,257.44,90.43,0.00),v40,z0,tPen\WObj:=wPaper;
    MoveL Offs(pOrigin,257.86,90.64,0.00),v40,fine,tPen\WObj:=wPaper;
    MoveL Offs(pOrigin,257.86,90.64,6.00),v60,z5,tPen\WObj:=wPaper;
    MoveL Offs(pOrigin,257.23,89.57,6.00),vTravel,z5,tPen\WObj:=wPaper;
    MoveL Offs(pOrigin,257.23,89.57,0.00),v60,z0,tPen\WObj:=wPaper;
    MoveL Offs(pOrigin,252.34,81.71,0.00),v40,fine,tPen\WObj:=wPaper;
    MoveL Offs(pOrigin,252.34,81.71,6.00),v60,z5,tPen\WObj:=wPaper;
    MoveL Offs(pOrigin,243.31,82.51,6.00),vTravel,z5,tPen\WObj:=wPaper;
    MoveL Offs(pOrigin,243.31,82.51,0.00),v60,z0,tPen\WObj:=wPaper;
    MoveL Offs(pOrigin,241.35,84.46,0.00),v40,fine,tPen\WObj:=wPaper;
    MoveL Offs(pOrigin,241.35,84.46,6.00),v60,z5,tPen\WObj:=wPaper;
    MoveL Offs(pOrigin,241.22,80.12,6.00),vTravel,z5,tPen\WObj:=wPaper;
    MoveL Offs(pOrigin,241.22,80.12,0.00),v60,z0,tPen\WObj:=wPaper;
    MoveL Offs(pOrigin,243.17,78.16,0.00),v40,fine,tPen\WObj:=wPaper;
    MoveL Offs(pOrigin,243.17,78.16,6.00),v60,z5,tPen\WObj:=wPaper;
    MoveL Offs(pOrigin,236.89,73.99,6.00),vTravel,z5,tPen\WObj:=wPaper;
    MoveL Offs(pOrigin,236.89,73.99,0.00),v60,z0,tPen\WObj:=wPaper;
    MoveL Offs(pOrigin,228.02,82.85,0.00),v40,fine,tPen\WObj:=wPaper;
    MoveL Offs(pOrigin,228.02,82.85,6.00),v60,z5,tPen\WObj:=wPaper;
    MoveL Offs(pOrigin,228.96,81.53,6.00),vTravel,z5,tPen\WObj:=wPaper;
    MoveL Offs(pOrigin,228.96,81.53,0.00),v60,z0,tPen\WObj:=wPaper;
    MoveL Offs(pOrigin,230.66,81.53,0.00),v40,z0,tPen\WObj:=wPaper;
    MoveL Offs(pOrigin,230.88,82.14,0.00),v40,z0,tPen\WObj:=wPaper;
    MoveL Offs(pOrigin,234.27,76.40,0.00),v40,z0,tPen\WObj:=wPaper;
    MoveL Offs(pOrigin,238.31,71.09,0.00),v40,fine,tPen\WObj:=wPaper;
    MoveL Offs(pOrigin,238.31,71.09,6.00),v60,z5,tPen\WObj:=wPaper;
    MoveL Offs(pOrigin,237.20,72.19,6.00),vTravel,z5,tPen\WObj:=wPaper;
    MoveL Offs(pOrigin,237.20,72.19,0.00),v60,z0,tPen\WObj:=wPaper;
    MoveL Offs(pOrigin,232.69,76.70,0.00),v40,fine,tPen\WObj:=wPaper;
    MoveL Offs(pOrigin,232.69,76.70,6.00),v60,z5,tPen\WObj:=wPaper;
    MoveL Offs(pOrigin,230.74,77.15,6.00),vTravel,z5,tPen\WObj:=wPaper;
    MoveL Offs(pOrigin,230.74,77.15,0.00),v60,z0,tPen\WObj:=wPaper;
    MoveL Offs(pOrigin,227.58,80.31,0.00),v40,z0,tPen\WObj:=wPaper;
    MoveL Offs(pOrigin,228.75,80.47,0.00),v40,z0,tPen\WObj:=wPaper;
    MoveL Offs(pOrigin,230.24,80.47,0.00),v40,z0,tPen\WObj:=wPaper;
    MoveL Offs(pOrigin,229.81,79.42,0.00),v40,z0,tPen\WObj:=wPaper;
    MoveL Offs(pOrigin,228.75,79.42,0.00),v40,fine,tPen\WObj:=wPaper;
    MoveL Offs(pOrigin,228.75,79.42,6.00),v60,z5,tPen\WObj:=wPaper;
    MoveL Offs(pOrigin,227.44,78.96,6.00),vTravel,z5,tPen\WObj:=wPaper;
    MoveL Offs(pOrigin,227.44,78.96,0.00),v60,z0,tPen\WObj:=wPaper;
    MoveL Offs(pOrigin,230.29,76.11,0.00),v40,z0,tPen\WObj:=wPaper;
    MoveL Offs(pOrigin,229.84,76.31,0.00),v40,z0,tPen\WObj:=wPaper;
    MoveL Offs(pOrigin,226.83,73.30,0.00),v40,z0,tPen\WObj:=wPaper;
    MoveL Offs(pOrigin,226.55,73.87,0.00),v40,z0,tPen\WObj:=wPaper;
    MoveL Offs(pOrigin,229.41,71.01,0.00),v40,z0,tPen\WObj:=wPaper;
    MoveL Offs(pOrigin,228.96,69.97,0.00),v40,z0,tPen\WObj:=wPaper;
    MoveL Offs(pOrigin,226.26,72.67,0.00),v40,z0,tPen\WObj:=wPaper;
    MoveL Offs(pOrigin,225.81,71.63,0.00),v40,z0,tPen\WObj:=wPaper;
    MoveL Offs(pOrigin,228.67,68.77,0.00),v40,z0,tPen\WObj:=wPaper;
    MoveL Offs(pOrigin,228.32,68.81,0.00),v40,z0,tPen\WObj:=wPaper;
    MoveL Offs(pOrigin,225.01,65.51,0.00),v40,z0,tPen\WObj:=wPaper;
    MoveL Offs(pOrigin,224.63,65.34,0.00),v40,z0,tPen\WObj:=wPaper;
    MoveL Offs(pOrigin,227.34,62.63,0.00),v40,z0,tPen\WObj:=wPaper;
    MoveL Offs(pOrigin,226.80,62.82,0.00),v40,z0,tPen\WObj:=wPaper;
    MoveL Offs(pOrigin,223.34,59.36,0.00),v40,z0,tPen\WObj:=wPaper;
    MoveL Offs(pOrigin,223.00,59.50,0.00),v40,z0,tPen\WObj:=wPaper;
    MoveL Offs(pOrigin,225.56,56.95,0.00),v40,z0,tPen\WObj:=wPaper;
    MoveL Offs(pOrigin,225.13,56.67,0.00),v40,z0,tPen\WObj:=wPaper;
    MoveL Offs(pOrigin,218.52,50.06,0.00),v40,z0,tPen\WObj:=wPaper;
    MoveL Offs(pOrigin,219.40,49.85,0.00),v40,z0,tPen\WObj:=wPaper;
    MoveL Offs(pOrigin,222.59,49.85,0.00),v40,z0,tPen\WObj:=wPaper;
    MoveL Offs(pOrigin,223.33,50.21,0.00),v40,z0,tPen\WObj:=wPaper;
    MoveL Offs(pOrigin,220.63,52.92,0.00),v40,z0,tPen\WObj:=wPaper;
    MoveL Offs(pOrigin,221.22,53.81,0.00),v40,z0,tPen\WObj:=wPaper;
    MoveL Offs(pOrigin,223.78,51.26,0.00),v40,z0,tPen\WObj:=wPaper;
    MoveL Offs(pOrigin,223.01,51.96,0.00),v40,z0,tPen\WObj:=wPaper;
    MoveL Offs(pOrigin,221.52,51.96,0.00),v40,z0,tPen\WObj:=wPaper;
    MoveL Offs(pOrigin,221.77,51.75,0.00),v40,z0,tPen\WObj:=wPaper;
    MoveL Offs(pOrigin,221.77,48.14,0.00),v40,z0,tPen\WObj:=wPaper;
    MoveL Offs(pOrigin,222.59,48.79,0.00),v40,z0,tPen\WObj:=wPaper;
  ENDPROC

  PROC DrawPart169()
    MoveL Offs(pOrigin,220.25,48.79,0.00),v40,z0,tPen\WObj:=wPaper;
    MoveL Offs(pOrigin,220.46,48.78,0.00),v40,z0,tPen\WObj:=wPaper;
    MoveL Offs(pOrigin,220.68,48.35,0.00),v40,z0,tPen\WObj:=wPaper;
    MoveL Offs(pOrigin,220.46,48.78,0.00),v40,z0,tPen\WObj:=wPaper;
    MoveL Offs(pOrigin,220.72,48.99,0.00),v40,z0,tPen\WObj:=wPaper;
    MoveL Offs(pOrigin,220.72,51.11,0.00),v40,fine,tPen\WObj:=wPaper;
    MoveL Offs(pOrigin,220.72,51.11,6.00),v60,z5,tPen\WObj:=wPaper;
    MoveL Offs(pOrigin,219.82,49.41,6.00),vTravel,z5,tPen\WObj:=wPaper;
    MoveL Offs(pOrigin,219.82,49.41,0.00),v60,z0,tPen\WObj:=wPaper;
    MoveL Offs(pOrigin,220.04,48.99,0.00),v40,z0,tPen\WObj:=wPaper;
    MoveL Offs(pOrigin,219.82,49.41,0.00),v40,z0,tPen\WObj:=wPaper;
    MoveL Offs(pOrigin,219.27,49.31,0.00),v40,z0,tPen\WObj:=wPaper;
    MoveL Offs(pOrigin,224.53,54.57,0.00),v40,z0,tPen\WObj:=wPaper;
    MoveL Offs(pOrigin,224.82,54.70,0.00),v40,z0,tPen\WObj:=wPaper;
    MoveL Offs(pOrigin,222.26,57.26,0.00),v40,z0,tPen\WObj:=wPaper;
    MoveL Offs(pOrigin,222.74,57.26,0.00),v40,z0,tPen\WObj:=wPaper;
    MoveL Offs(pOrigin,226.34,60.87,0.00),v40,z0,tPen\WObj:=wPaper;
    MoveL Offs(pOrigin,226.60,60.39,0.00),v40,z0,tPen\WObj:=wPaper;
    MoveL Offs(pOrigin,223.89,63.09,0.00),v40,z0,tPen\WObj:=wPaper;
    MoveL Offs(pOrigin,224.92,62.52,0.00),v40,z0,tPen\WObj:=wPaper;
    MoveL Offs(pOrigin,226.20,62.52,0.00),v40,z0,tPen\WObj:=wPaper;
    MoveL Offs(pOrigin,225.99,61.46,0.00),v40,z0,tPen\WObj:=wPaper;
    MoveL Offs(pOrigin,224.71,61.46,0.00),v40,z0,tPen\WObj:=wPaper;
    MoveL Offs(pOrigin,224.94,61.52,0.00),v40,z0,tPen\WObj:=wPaper;
    MoveL Offs(pOrigin,224.94,60.46,0.00),v40,z0,tPen\WObj:=wPaper;
    MoveL Offs(pOrigin,225.56,60.41,0.00),v40,z0,tPen\WObj:=wPaper;
    MoveL Offs(pOrigin,224.29,60.41,0.00),v40,z0,tPen\WObj:=wPaper;
    MoveL Offs(pOrigin,224.08,59.35,0.00),v40,z0,tPen\WObj:=wPaper;
    MoveL Offs(pOrigin,225.35,59.35,0.00),v40,z0,tPen\WObj:=wPaper;
    MoveL Offs(pOrigin,226.30,59.19,0.00),v40,z0,tPen\WObj:=wPaper;
    MoveL Offs(pOrigin,223.60,61.90,0.00),v40,fine,tPen\WObj:=wPaper;
    MoveL Offs(pOrigin,223.60,61.90,6.00),v60,z5,tPen\WObj:=wPaper;
    MoveL Offs(pOrigin,224.19,64.29,6.00),vTravel,z5,tPen\WObj:=wPaper;
    MoveL Offs(pOrigin,224.19,64.29,0.00),v60,z0,tPen\WObj:=wPaper;
    MoveL Offs(pOrigin,226.89,61.59,0.00),v40,fine,tPen\WObj:=wPaper;
    MoveL Offs(pOrigin,226.89,61.59,6.00),v60,z5,tPen\WObj:=wPaper;
    MoveL Offs(pOrigin,227.05,64.63,6.00),vTravel,z5,tPen\WObj:=wPaper;
    MoveL Offs(pOrigin,227.05,64.63,0.00),v60,z0,tPen\WObj:=wPaper;
    MoveL Offs(pOrigin,225.35,64.63,0.00),v40,fine,tPen\WObj:=wPaper;
    MoveL Offs(pOrigin,225.35,64.63,6.00),v60,z5,tPen\WObj:=wPaper;
    MoveL Offs(pOrigin,227.26,65.14,6.00),vTravel,z5,tPen\WObj:=wPaper;
    MoveL Offs(pOrigin,227.26,65.14,0.00),v60,z0,tPen\WObj:=wPaper;
    MoveL Offs(pOrigin,227.26,66.62,0.00),v40,z0,tPen\WObj:=wPaper;
    MoveL Offs(pOrigin,227.69,67.05,0.00),v40,z0,tPen\WObj:=wPaper;
    MoveL Offs(pOrigin,227.69,67.05,0.00),v40,z0,tPen\WObj:=wPaper;
    MoveL Offs(pOrigin,228.75,66.91,0.00),v40,z0,tPen\WObj:=wPaper;
    MoveL Offs(pOrigin,233.00,64.78,0.00),v40,z0,tPen\WObj:=wPaper;
    MoveL Offs(pOrigin,235.76,62.80,0.00),v40,z0,tPen\WObj:=wPaper;
    MoveL Offs(pOrigin,237.25,61.10,0.00),v40,z0,tPen\WObj:=wPaper;
    MoveL Offs(pOrigin,236.93,62.00,0.00),v40,z0,tPen\WObj:=wPaper;
    MoveL Offs(pOrigin,232.87,66.06,0.00),v40,fine,tPen\WObj:=wPaper;
    MoveL Offs(pOrigin,232.87,66.06,6.00),v60,z5,tPen\WObj:=wPaper;
    MoveL Offs(pOrigin,230.32,67.12,6.00),vTravel,z5,tPen\WObj:=wPaper;
    MoveL Offs(pOrigin,230.32,67.12,0.00),v60,z0,tPen\WObj:=wPaper;
    MoveL Offs(pOrigin,235.88,61.56,0.00),v40,fine,tPen\WObj:=wPaper;
    MoveL Offs(pOrigin,235.88,61.56,6.00),v60,z5,tPen\WObj:=wPaper;
    MoveL Offs(pOrigin,240.29,64.36,6.00),vTravel,z5,tPen\WObj:=wPaper;
    MoveL Offs(pOrigin,240.29,64.36,0.00),v60,z0,tPen\WObj:=wPaper;
    MoveL Offs(pOrigin,241.19,65.26,0.00),v40,z0,tPen\WObj:=wPaper;
    MoveL Offs(pOrigin,241.86,64.54,0.00),v40,z0,tPen\WObj:=wPaper;
    MoveL Offs(pOrigin,239.91,66.49,0.00),v40,fine,tPen\WObj:=wPaper;
    MoveL Offs(pOrigin,239.91,66.49,6.00),v60,z5,tPen\WObj:=wPaper;
    MoveL Offs(pOrigin,240.60,67.65,6.00),vTravel,z5,tPen\WObj:=wPaper;
    MoveL Offs(pOrigin,240.60,67.65,0.00),v60,z0,tPen\WObj:=wPaper;
    MoveL Offs(pOrigin,241.50,68.55,0.00),v40,z0,tPen\WObj:=wPaper;
    MoveL Offs(pOrigin,242.15,68.73,0.00),v40,z0,tPen\WObj:=wPaper;
    MoveL Offs(pOrigin,240.35,70.53,0.00),v40,fine,tPen\WObj:=wPaper;
    MoveL Offs(pOrigin,240.35,70.53,6.00),v60,z5,tPen\WObj:=wPaper;
    MoveL Offs(pOrigin,239.90,67.99,6.00),vTravel,z5,tPen\WObj:=wPaper;
    MoveL Offs(pOrigin,239.90,67.99,0.00),v60,z0,tPen\WObj:=wPaper;
    MoveL Offs(pOrigin,242.01,65.88,0.00),v40,fine,tPen\WObj:=wPaper;
    MoveL Offs(pOrigin,242.01,65.88,6.00),v60,z5,tPen\WObj:=wPaper;
    MoveL Offs(pOrigin,244.55,67.82,6.00),vTravel,z5,tPen\WObj:=wPaper;
    MoveL Offs(pOrigin,244.55,67.82,0.00),v60,z0,tPen\WObj:=wPaper;
    MoveL Offs(pOrigin,247.70,64.67,0.00),v40,z0,tPen\WObj:=wPaper;
    MoveL Offs(pOrigin,248.09,65.56,0.00),v40,z0,tPen\WObj:=wPaper;
    MoveL Offs(pOrigin,246.60,66.20,0.00),v40,z0,tPen\WObj:=wPaper;
    MoveL Offs(pOrigin,245.61,68.11,0.00),v40,z0,tPen\WObj:=wPaper;
    MoveL Offs(pOrigin,246.18,70.03,0.00),v40,z0,tPen\WObj:=wPaper;
    MoveL Offs(pOrigin,247.66,71.09,0.00),v40,z0,tPen\WObj:=wPaper;
    MoveL Offs(pOrigin,249.36,71.09,0.00),v40,z0,tPen\WObj:=wPaper;
    MoveL Offs(pOrigin,250.43,70.45,0.00),v40,z0,tPen\WObj:=wPaper;
    MoveL Offs(pOrigin,251.27,68.96,0.00),v40,z0,tPen\WObj:=wPaper;
    MoveL Offs(pOrigin,251.27,67.69,0.00),v40,z0,tPen\WObj:=wPaper;
    MoveL Offs(pOrigin,250.85,66.84,0.00),v40,z0,tPen\WObj:=wPaper;
    MoveL Offs(pOrigin,249.79,65.85,0.00),v40,z0,tPen\WObj:=wPaper;
    MoveL Offs(pOrigin,248.09,65.56,0.00),v40,z0,tPen\WObj:=wPaper;
    MoveL Offs(pOrigin,248.98,65.58,0.00),v40,z0,tPen\WObj:=wPaper;
    MoveL Offs(pOrigin,250.93,67.53,0.00),v40,z0,tPen\WObj:=wPaper;
    MoveL Offs(pOrigin,252.04,67.80,0.00),v40,z0,tPen\WObj:=wPaper;
    MoveL Offs(pOrigin,247.98,71.86,0.00),v40,z0,tPen\WObj:=wPaper;
    MoveL Offs(pOrigin,246.93,71.41,0.00),v40,z0,tPen\WObj:=wPaper;
    MoveL Offs(pOrigin,251.74,66.60,0.00),v40,z0,tPen\WObj:=wPaper;
    MoveL Offs(pOrigin,251.00,65.86,0.00),v40,z0,tPen\WObj:=wPaper;
    MoveL Offs(pOrigin,245.89,70.96,0.00),v40,z0,tPen\WObj:=wPaper;
    MoveL Offs(pOrigin,245.29,70.07,0.00),v40,z0,tPen\WObj:=wPaper;
    MoveL Offs(pOrigin,250.25,65.11,0.00),v40,z0,tPen\WObj:=wPaper;
    MoveL Offs(pOrigin,249.20,64.66,0.00),v40,z0,tPen\WObj:=wPaper;
    MoveL Offs(pOrigin,244.84,69.02,0.00),v40,fine,tPen\WObj:=wPaper;
    MoveL Offs(pOrigin,244.84,69.02,6.00),v60,z5,tPen\WObj:=wPaper;
    MoveL Offs(pOrigin,247.88,67.90,6.00),vTravel,z5,tPen\WObj:=wPaper;
    MoveL Offs(pOrigin,247.88,67.90,0.00),v60,z0,tPen\WObj:=wPaper;
    MoveL Offs(pOrigin,247.95,68.75,0.00),v40,z0,tPen\WObj:=wPaper;
    MoveL Offs(pOrigin,248.30,68.96,0.00),v40,z0,tPen\WObj:=wPaper;
    MoveL Offs(pOrigin,249.08,68.89,0.00),v40,z0,tPen\WObj:=wPaper;
    MoveL Offs(pOrigin,249.15,68.11,0.00),v40,fine,tPen\WObj:=wPaper;
    MoveL Offs(pOrigin,249.15,68.11,6.00),v60,z5,tPen\WObj:=wPaper;
    MoveL Offs(pOrigin,252.03,69.30,6.00),vTravel,z5,tPen\WObj:=wPaper;
    MoveL Offs(pOrigin,252.03,69.30,0.00),v60,z0,tPen\WObj:=wPaper;
    MoveL Offs(pOrigin,249.63,71.70,0.00),v40,fine,tPen\WObj:=wPaper;
    MoveL Offs(pOrigin,249.63,71.70,6.00),v60,z5,tPen\WObj:=wPaper;
    MoveL Offs(pOrigin,260.28,67.03,6.00),vTravel,z5,tPen\WObj:=wPaper;
    MoveL Offs(pOrigin,260.28,67.03,0.00),v60,z0,tPen\WObj:=wPaper;
    MoveL Offs(pOrigin,261.18,66.12,0.00),v40,z0,tPen\WObj:=wPaper;
    MoveL Offs(pOrigin,262.08,66.72,0.00),v40,z0,tPen\WObj:=wPaper;
    MoveL Offs(pOrigin,261.03,67.77,0.00),v40,z0,tPen\WObj:=wPaper;
    MoveL Offs(pOrigin,261.62,68.67,0.00),v40,z0,tPen\WObj:=wPaper;
    MoveL Offs(pOrigin,262.83,67.47,0.00),v40,z0,tPen\WObj:=wPaper;
    MoveL Offs(pOrigin,263.57,68.21,0.00),v40,z0,tPen\WObj:=wPaper;
    MoveL Offs(pOrigin,262.37,69.42,0.00),v40,z0,tPen\WObj:=wPaper;
  ENDPROC

  PROC DrawPart170()
    MoveL Offs(pOrigin,262.97,70.31,0.00),v40,z0,tPen\WObj:=wPaper;
    MoveL Offs(pOrigin,264.17,69.11,0.00),v40,z0,tPen\WObj:=wPaper;
    MoveL Offs(pOrigin,265.07,69.71,0.00),v40,z0,tPen\WObj:=wPaper;
    MoveL Offs(pOrigin,263.71,71.06,0.00),v40,z0,tPen\WObj:=wPaper;
    MoveL Offs(pOrigin,264.46,71.81,0.00),v40,z0,tPen\WObj:=wPaper;
    MoveL Offs(pOrigin,265.81,70.45,0.00),v40,z0,tPen\WObj:=wPaper;
    MoveL Offs(pOrigin,266.56,71.20,0.00),v40,z0,tPen\WObj:=wPaper;
    MoveL Offs(pOrigin,263.40,74.36,0.00),v40,z0,tPen\WObj:=wPaper;
    MoveL Offs(pOrigin,263.85,75.40,0.00),v40,z0,tPen\WObj:=wPaper;
    MoveL Offs(pOrigin,267.31,71.95,0.00),v40,z0,tPen\WObj:=wPaper;
    MoveL Offs(pOrigin,267.90,72.84,0.00),v40,z0,tPen\WObj:=wPaper;
    MoveL Offs(pOrigin,264.45,76.30,0.00),v40,z0,tPen\WObj:=wPaper;
    MoveL Offs(pOrigin,265.19,77.05,0.00),v40,z0,tPen\WObj:=wPaper;
    MoveL Offs(pOrigin,268.65,73.59,0.00),v40,z0,tPen\WObj:=wPaper;
    MoveL Offs(pOrigin,269.25,74.49,0.00),v40,z0,tPen\WObj:=wPaper;
    MoveL Offs(pOrigin,267.74,75.99,0.00),v40,z0,tPen\WObj:=wPaper;
    MoveL Offs(pOrigin,268.48,76.13,0.00),v40,z0,tPen\WObj:=wPaper;
    MoveL Offs(pOrigin,273.89,81.54,0.00),v40,z0,tPen\WObj:=wPaper;
    MoveL Offs(pOrigin,273.38,81.53,0.00),v40,z0,tPen\WObj:=wPaper;
    MoveL Offs(pOrigin,272.10,81.53,0.00),v40,z0,tPen\WObj:=wPaper;
    MoveL Offs(pOrigin,272.46,81.50,0.00),v40,z0,tPen\WObj:=wPaper;
    MoveL Offs(pOrigin,272.46,79.38,0.00),v40,z0,tPen\WObj:=wPaper;
    MoveL Offs(pOrigin,271.89,79.42,0.00),v40,z0,tPen\WObj:=wPaper;
    MoveL Offs(pOrigin,273.59,79.42,0.00),v40,z0,tPen\WObj:=wPaper;
    MoveL Offs(pOrigin,274.62,79.56,0.00),v40,z0,tPen\WObj:=wPaper;
    MoveL Offs(pOrigin,270.72,83.47,0.00),v40,fine,tPen\WObj:=wPaper;
    MoveL Offs(pOrigin,270.72,83.47,6.00),v60,z5,tPen\WObj:=wPaper;
    MoveL Offs(pOrigin,271.06,84.67,6.00),vTravel,z5,tPen\WObj:=wPaper;
    MoveL Offs(pOrigin,271.06,84.67,0.00),v60,z0,tPen\WObj:=wPaper;
    MoveL Offs(pOrigin,273.31,86.93,0.00),v40,z0,tPen\WObj:=wPaper;
    MoveL Offs(pOrigin,274.00,86.16,0.00),v40,z0,tPen\WObj:=wPaper;
    MoveL Offs(pOrigin,270.10,90.06,0.00),v40,z0,tPen\WObj:=wPaper;
    MoveL Offs(pOrigin,270.62,90.21,0.00),v40,z0,tPen\WObj:=wPaper;
    MoveL Offs(pOrigin,272.73,92.32,0.00),v40,z0,tPen\WObj:=wPaper;
    MoveL Offs(pOrigin,272.31,92.09,0.00),v40,z0,tPen\WObj:=wPaper;
    MoveL Offs(pOrigin,271.04,92.09,0.00),v40,z0,tPen\WObj:=wPaper;
    MoveL Offs(pOrigin,271.04,93.14,0.00),v40,z0,tPen\WObj:=wPaper;
    MoveL Offs(pOrigin,272.10,93.14,0.00),v40,fine,tPen\WObj:=wPaper;
    MoveL Offs(pOrigin,272.10,93.14,6.00),v60,z5,tPen\WObj:=wPaper;
    MoveL Offs(pOrigin,273.38,92.75,6.00),vTravel,z5,tPen\WObj:=wPaper;
    MoveL Offs(pOrigin,273.38,92.75,0.00),v60,z0,tPen\WObj:=wPaper;
    MoveL Offs(pOrigin,269.63,96.51,0.00),v40,z0,tPen\WObj:=wPaper;
    MoveL Offs(pOrigin,270.05,97.10,0.00),v40,z0,tPen\WObj:=wPaper;
    MoveL Offs(pOrigin,272.30,99.36,0.00),v40,z0,tPen\WObj:=wPaper;
    MoveL Offs(pOrigin,271.89,99.48,0.00),v40,z0,tPen\WObj:=wPaper;
    MoveL Offs(pOrigin,270.82,99.48,0.00),v40,z0,tPen\WObj:=wPaper;
    MoveL Offs(pOrigin,270.82,98.42,0.00),v40,z0,tPen\WObj:=wPaper;
    MoveL Offs(pOrigin,271.89,98.42,0.00),v40,z0,tPen\WObj:=wPaper;
    MoveL Offs(pOrigin,271.89,97.37,0.00),v40,z0,tPen\WObj:=wPaper;
    MoveL Offs(pOrigin,270.82,97.37,0.00),v40,fine,tPen\WObj:=wPaper;
    MoveL Offs(pOrigin,270.82,97.37,6.00),v60,z5,tPen\WObj:=wPaper;
    MoveL Offs(pOrigin,270.82,95.26,6.00),vTravel,z5,tPen\WObj:=wPaper;
    MoveL Offs(pOrigin,270.82,95.26,0.00),v60,z0,tPen\WObj:=wPaper;
    MoveL Offs(pOrigin,272.10,95.26,0.00),v40,fine,tPen\WObj:=wPaper;
    MoveL Offs(pOrigin,272.10,95.26,6.00),v60,z5,tPen\WObj:=wPaper;
    MoveL Offs(pOrigin,273.07,96.05,6.00),vTravel,z5,tPen\WObj:=wPaper;
    MoveL Offs(pOrigin,273.07,96.05,0.00),v60,z0,tPen\WObj:=wPaper;
    MoveL Offs(pOrigin,269.47,99.65,0.00),v40,fine,tPen\WObj:=wPaper;
    MoveL Offs(pOrigin,269.47,99.65,6.00),v60,z5,tPen\WObj:=wPaper;
    MoveL Offs(pOrigin,270.61,101.59,6.00),vTravel,z5,tPen\WObj:=wPaper;
    MoveL Offs(pOrigin,270.61,101.59,0.00),v60,z0,tPen\WObj:=wPaper;
    MoveL Offs(pOrigin,271.68,101.59,0.00),v40,z0,tPen\WObj:=wPaper;
    MoveL Offs(pOrigin,271.68,102.65,0.00),v40,z0,tPen\WObj:=wPaper;
    MoveL Offs(pOrigin,270.61,102.65,0.00),v40,z0,tPen\WObj:=wPaper;
    MoveL Offs(pOrigin,269.91,102.95,0.00),v40,z0,tPen\WObj:=wPaper;
    MoveL Offs(pOrigin,272.32,105.35,0.00),v40,z0,tPen\WObj:=wPaper;
    MoveL Offs(pOrigin,272.75,105.34,0.00),v40,z0,tPen\WObj:=wPaper;
    MoveL Offs(pOrigin,269.44,108.64,0.00),v40,z0,tPen\WObj:=wPaper;
    MoveL Offs(pOrigin,269.93,108.94,0.00),v40,z0,tPen\WObj:=wPaper;
    MoveL Offs(pOrigin,272.34,111.34,0.00),v40,z0,tPen\WObj:=wPaper;
    MoveL Offs(pOrigin,272.88,111.18,0.00),v40,z0,tPen\WObj:=wPaper;
    MoveL Offs(pOrigin,268.52,115.54,0.00),v40,z0,tPen\WObj:=wPaper;
    MoveL Offs(pOrigin,267.92,114.64,0.00),v40,z0,tPen\WObj:=wPaper;
    MoveL Offs(pOrigin,272.73,109.83,0.00),v40,fine,tPen\WObj:=wPaper;
    MoveL Offs(pOrigin,272.73,109.83,6.00),v60,z5,tPen\WObj:=wPaper;
    MoveL Offs(pOrigin,271.68,108.98,6.00),vTravel,z5,tPen\WObj:=wPaper;
    MoveL Offs(pOrigin,271.68,108.98,0.00),v60,z0,tPen\WObj:=wPaper;
    MoveL Offs(pOrigin,270.61,108.98,0.00),v40,z0,tPen\WObj:=wPaper;
    MoveL Offs(pOrigin,270.61,107.93,0.00),v40,z0,tPen\WObj:=wPaper;
    MoveL Offs(pOrigin,271.68,107.93,0.00),v40,z0,tPen\WObj:=wPaper;
    MoveL Offs(pOrigin,271.68,106.87,0.00),v40,z0,tPen\WObj:=wPaper;
    MoveL Offs(pOrigin,270.61,106.87,0.00),v40,z0,tPen\WObj:=wPaper;
    MoveL Offs(pOrigin,270.61,105.82,0.00),v40,z0,tPen\WObj:=wPaper;
    MoveL Offs(pOrigin,271.68,105.82,0.00),v40,z0,tPen\WObj:=wPaper;
    MoveL Offs(pOrigin,271.68,104.76,0.00),v40,z0,tPen\WObj:=wPaper;
    MoveL Offs(pOrigin,270.61,104.76,0.00),v40,z0,tPen\WObj:=wPaper;
    MoveL Offs(pOrigin,269.92,104.44,0.00),v40,z0,tPen\WObj:=wPaper;
    MoveL Offs(pOrigin,272.32,106.85,0.00),v40,z0,tPen\WObj:=wPaper;
    MoveL Offs(pOrigin,272.74,106.83,0.00),v40,z0,tPen\WObj:=wPaper;
    MoveL Offs(pOrigin,269.44,110.14,0.00),v40,fine,tPen\WObj:=wPaper;
    MoveL Offs(pOrigin,269.44,110.14,6.00),v60,z5,tPen\WObj:=wPaper;
    MoveL Offs(pOrigin,267.79,110.29,6.00),vTravel,z5,tPen\WObj:=wPaper;
    MoveL Offs(pOrigin,267.79,110.29,0.00),v60,z0,tPen\WObj:=wPaper;
    MoveL Offs(pOrigin,266.43,111.65,0.00),v40,z0,tPen\WObj:=wPaper;
    MoveL Offs(pOrigin,265.99,110.60,0.00),v40,z0,tPen\WObj:=wPaper;
    MoveL Offs(pOrigin,267.34,109.25,0.00),v40,z0,tPen\WObj:=wPaper;
    MoveL Offs(pOrigin,266.89,108.20,0.00),v40,z0,tPen\WObj:=wPaper;
    MoveL Offs(pOrigin,265.54,109.55,0.00),v40,z0,tPen\WObj:=wPaper;
    MoveL Offs(pOrigin,265.10,108.51,0.00),v40,z0,tPen\WObj:=wPaper;
    MoveL Offs(pOrigin,266.60,107.00,0.00),v40,z0,tPen\WObj:=wPaper;
    MoveL Offs(pOrigin,266.15,105.96,0.00),v40,z0,tPen\WObj:=wPaper;
    MoveL Offs(pOrigin,264.80,107.31,0.00),v40,z0,tPen\WObj:=wPaper;
    MoveL Offs(pOrigin,264.20,106.41,0.00),v40,z0,tPen\WObj:=wPaper;
    MoveL Offs(pOrigin,265.71,104.91,0.00),v40,z0,tPen\WObj:=wPaper;
    MoveL Offs(pOrigin,265.26,103.86,0.00),v40,z0,tPen\WObj:=wPaper;
    MoveL Offs(pOrigin,263.76,105.36,0.00),v40,z0,tPen\WObj:=wPaper;
    MoveL Offs(pOrigin,263.31,104.32,0.00),v40,z0,tPen\WObj:=wPaper;
    MoveL Offs(pOrigin,264.81,102.81,0.00),v40,z0,tPen\WObj:=wPaper;
    MoveL Offs(pOrigin,264.37,101.77,0.00),v40,z0,tPen\WObj:=wPaper;
    MoveL Offs(pOrigin,262.87,103.27,0.00),v40,z0,tPen\WObj:=wPaper;
    MoveL Offs(pOrigin,262.27,102.37,0.00),v40,z0,tPen\WObj:=wPaper;
    MoveL Offs(pOrigin,263.92,100.72,0.00),v40,z0,tPen\WObj:=wPaper;
    MoveL Offs(pOrigin,263.33,99.82,0.00),v40,z0,tPen\WObj:=wPaper;
    MoveL Offs(pOrigin,261.97,101.17,0.00),v40,z0,tPen\WObj:=wPaper;
    MoveL Offs(pOrigin,261.38,100.28,0.00),v40,z0,tPen\WObj:=wPaper;
    MoveL Offs(pOrigin,262.88,98.77,0.00),v40,z0,tPen\WObj:=wPaper;
    MoveL Offs(pOrigin,262.11,99.14,0.00),v40,z0,tPen\WObj:=wPaper;
    MoveL Offs(pOrigin,262.33,99.56,0.00),v40,z0,tPen\WObj:=wPaper;
    MoveL Offs(pOrigin,262.11,99.14,0.00),v40,fine,tPen\WObj:=wPaper;
    MoveL Offs(pOrigin,262.11,99.14,6.00),v60,z5,tPen\WObj:=wPaper;
  ENDPROC

  PROC DrawPart171()
    MoveL Offs(pOrigin,269.46,102.65,6.00),vTravel,z5,tPen\WObj:=wPaper;
    MoveL Offs(pOrigin,269.46,102.65,0.00),v60,z0,tPen\WObj:=wPaper;
    MoveL Offs(pOrigin,272.91,99.19,0.00),v40,fine,tPen\WObj:=wPaper;
    MoveL Offs(pOrigin,272.91,99.19,6.00),v60,z5,tPen\WObj:=wPaper;
    MoveL Offs(pOrigin,272.91,100.69,6.00),vTravel,z5,tPen\WObj:=wPaper;
    MoveL Offs(pOrigin,272.91,100.69,0.00),v60,z0,tPen\WObj:=wPaper;
    MoveL Offs(pOrigin,269.45,104.15,0.00),v40,fine,tPen\WObj:=wPaper;
    MoveL Offs(pOrigin,269.45,104.15,6.00),v60,z5,tPen\WObj:=wPaper;
    MoveL Offs(pOrigin,270.61,103.70,6.00),vTravel,z5,tPen\WObj:=wPaper;
    MoveL Offs(pOrigin,270.61,103.70,0.00),v60,z0,tPen\WObj:=wPaper;
    MoveL Offs(pOrigin,271.68,103.70,0.00),v40,fine,tPen\WObj:=wPaper;
    MoveL Offs(pOrigin,271.68,103.70,6.00),v60,z5,tPen\WObj:=wPaper;
    MoveL Offs(pOrigin,268.23,111.34,6.00),vTravel,z5,tPen\WObj:=wPaper;
    MoveL Offs(pOrigin,268.23,111.34,0.00),v60,z0,tPen\WObj:=wPaper;
    MoveL Offs(pOrigin,266.88,112.69,0.00),v40,z0,tPen\WObj:=wPaper;
    MoveL Offs(pOrigin,267.33,113.74,0.00),v40,z0,tPen\WObj:=wPaper;
    MoveL Offs(pOrigin,268.68,112.39,0.00),v40,fine,tPen\WObj:=wPaper;
    MoveL Offs(pOrigin,268.68,112.39,6.00),v60,z5,tPen\WObj:=wPaper;
    MoveL Offs(pOrigin,259.96,122.60,6.00),vTravel,z5,tPen\WObj:=wPaper;
    MoveL Offs(pOrigin,259.96,122.60,0.00),v60,z0,tPen\WObj:=wPaper;
    MoveL Offs(pOrigin,259.21,123.35,0.00),v40,z0,tPen\WObj:=wPaper;
    MoveL Offs(pOrigin,259.96,124.10,0.00),v40,z0,tPen\WObj:=wPaper;
    MoveL Offs(pOrigin,259.20,124.85,0.00),v40,z0,tPen\WObj:=wPaper;
    MoveL Offs(pOrigin,260.10,125.45,0.00),v40,z0,tPen\WObj:=wPaper;
    MoveL Offs(pOrigin,259.35,126.20,0.00),v40,z0,tPen\WObj:=wPaper;
    MoveL Offs(pOrigin,260.10,126.95,0.00),v40,z0,tPen\WObj:=wPaper;
    MoveL Offs(pOrigin,259.35,127.70,0.00),v40,z0,tPen\WObj:=wPaper;
    MoveL Offs(pOrigin,260.09,128.44,0.00),v40,z0,tPen\WObj:=wPaper;
    MoveL Offs(pOrigin,259.34,129.20,0.00),v40,fine,tPen\WObj:=wPaper;
    MoveL Offs(pOrigin,259.34,129.20,6.00),v60,z5,tPen\WObj:=wPaper;
    MoveL Offs(pOrigin,270.73,128.26,6.00),vTravel,z5,tPen\WObj:=wPaper;
    MoveL Offs(pOrigin,270.73,128.26,0.00),v60,z0,tPen\WObj:=wPaper;
    MoveL Offs(pOrigin,273.88,125.11,0.00),v40,fine,tPen\WObj:=wPaper;
    MoveL Offs(pOrigin,273.88,125.11,6.00),v60,z5,tPen\WObj:=wPaper;
    MoveL Offs(pOrigin,272.74,125.88,6.00),vTravel,z5,tPen\WObj:=wPaper;
    MoveL Offs(pOrigin,272.74,125.88,0.00),v60,z0,tPen\WObj:=wPaper;
    MoveL Offs(pOrigin,271.68,125.88,0.00),v40,fine,tPen\WObj:=wPaper;
    MoveL Offs(pOrigin,271.68,125.88,6.00),v60,z5,tPen\WObj:=wPaper;
    MoveL Offs(pOrigin,271.89,127.99,6.00),vTravel,z5,tPen\WObj:=wPaper;
    MoveL Offs(pOrigin,271.89,127.99,0.00),v60,z0,tPen\WObj:=wPaper;
    MoveL Offs(pOrigin,272.95,127.99,0.00),v40,z0,tPen\WObj:=wPaper;
    MoveL Offs(pOrigin,273.16,129.05,0.00),v40,z0,tPen\WObj:=wPaper;
    MoveL Offs(pOrigin,272.10,129.05,0.00),v40,fine,tPen\WObj:=wPaper;
    MoveL Offs(pOrigin,272.10,129.05,6.00),v60,z5,tPen\WObj:=wPaper;
    MoveL Offs(pOrigin,271.04,127.97,6.00),vTravel,z5,tPen\WObj:=wPaper;
    MoveL Offs(pOrigin,271.04,127.97,0.00),v60,z0,tPen\WObj:=wPaper;
    MoveL Offs(pOrigin,273.74,130.67,0.00),v40,z0,tPen\WObj:=wPaper;
    MoveL Offs(pOrigin,273.38,131.16,0.00),v40,z0,tPen\WObj:=wPaper;
    MoveL Offs(pOrigin,272.31,131.16,0.00),v40,fine,tPen\WObj:=wPaper;
    MoveL Offs(pOrigin,272.31,131.16,6.00),v60,z5,tPen\WObj:=wPaper;
    MoveL Offs(pOrigin,272.52,133.27,6.00),vTravel,z5,tPen\WObj:=wPaper;
    MoveL Offs(pOrigin,272.52,133.27,0.00),v60,z0,tPen\WObj:=wPaper;
    MoveL Offs(pOrigin,273.59,133.27,0.00),v40,z0,tPen\WObj:=wPaper;
    MoveL Offs(pOrigin,273.80,134.33,0.00),v40,z0,tPen\WObj:=wPaper;
    MoveL Offs(pOrigin,272.74,134.33,0.00),v40,fine,tPen\WObj:=wPaper;
    MoveL Offs(pOrigin,272.74,134.33,6.00),v60,z5,tPen\WObj:=wPaper;
    MoveL Offs(pOrigin,271.46,133.50,6.00),vTravel,z5,tPen\WObj:=wPaper;
    MoveL Offs(pOrigin,271.46,133.50,0.00),v60,z0,tPen\WObj:=wPaper;
    MoveL Offs(pOrigin,274.47,130.50,0.00),v40,fine,tPen\WObj:=wPaper;
    MoveL Offs(pOrigin,274.47,130.50,6.00),v60,z5,tPen\WObj:=wPaper;
    MoveL Offs(pOrigin,274.90,134.54,6.00),vTravel,z5,tPen\WObj:=wPaper;
    MoveL Offs(pOrigin,274.90,134.54,0.00),v60,z0,tPen\WObj:=wPaper;
    MoveL Offs(pOrigin,272.05,137.40,0.00),v40,z0,tPen\WObj:=wPaper;
    MoveL Offs(pOrigin,273.16,137.50,0.00),v40,z0,tPen\WObj:=wPaper;
    MoveL Offs(pOrigin,274.23,137.50,0.00),v40,z0,tPen\WObj:=wPaper;
    MoveL Offs(pOrigin,274.01,136.44,0.00),v40,z0,tPen\WObj:=wPaper;
    MoveL Offs(pOrigin,272.95,136.44,0.00),v40,fine,tPen\WObj:=wPaper;
    MoveL Offs(pOrigin,272.95,136.44,6.00),v60,z5,tPen\WObj:=wPaper;
    MoveL Offs(pOrigin,268.70,156.94,6.00),vTravel,z5,tPen\WObj:=wPaper;
    MoveL Offs(pOrigin,268.70,156.94,0.00),v60,z0,tPen\WObj:=wPaper;
    MoveL Offs(pOrigin,271.82,165.44,0.00),v40,z0,tPen\WObj:=wPaper;
    MoveL Offs(pOrigin,276.21,175.00,0.00),v40,z0,tPen\WObj:=wPaper;
    MoveL Offs(pOrigin,276.56,176.70,0.00),v40,z0,tPen\WObj:=wPaper;
    MoveL Offs(pOrigin,276.58,176.82,0.00),v40,z0,tPen\WObj:=wPaper;
    MoveL Offs(pOrigin,279.74,179.97,0.00),v40,z0,tPen\WObj:=wPaper;
    MoveL Offs(pOrigin,279.11,179.74,0.00),v40,z0,tPen\WObj:=wPaper;
    MoveL Offs(pOrigin,277.84,179.74,0.00),v40,z0,tPen\WObj:=wPaper;
    MoveL Offs(pOrigin,276.89,180.11,0.00),v40,z0,tPen\WObj:=wPaper;
    MoveL Offs(pOrigin,279.15,182.37,0.00),v40,z0,tPen\WObj:=wPaper;
    MoveL Offs(pOrigin,278.48,181.85,0.00),v40,z0,tPen\WObj:=wPaper;
    MoveL Offs(pOrigin,277.41,181.85,0.00),v40,z0,tPen\WObj:=wPaper;
    MoveL Offs(pOrigin,277.20,181.16,0.00),v40,z0,tPen\WObj:=wPaper;
    MoveL Offs(pOrigin,270.40,177.20,0.00),v40,z0,tPen\WObj:=wPaper;
    MoveL Offs(pOrigin,269.34,176.27,0.00),v40,z0,tPen\WObj:=wPaper;
    MoveL Offs(pOrigin,269.34,176.27,0.00),v40,z0,tPen\WObj:=wPaper;
    MoveL Offs(pOrigin,269.05,175.00,0.00),v40,z0,tPen\WObj:=wPaper;
    MoveL Offs(pOrigin,267.21,172.24,0.00),v40,z0,tPen\WObj:=wPaper;
    MoveL Offs(pOrigin,262.75,167.14,0.00),v40,z0,tPen\WObj:=wPaper;
    MoveL Offs(pOrigin,262.33,166.29,0.00),v40,z0,tPen\WObj:=wPaper;
    MoveL Offs(pOrigin,261.05,165.65,0.00),v40,z0,tPen\WObj:=wPaper;
    MoveL Offs(pOrigin,253.19,159.70,0.00),v40,z0,tPen\WObj:=wPaper;
    MoveL Offs(pOrigin,252.20,160.23,0.00),v40,z0,tPen\WObj:=wPaper;
    MoveL Offs(pOrigin,249.95,162.48,0.00),v40,z0,tPen\WObj:=wPaper;
    MoveL Offs(pOrigin,250.85,162.04,0.00),v40,z0,tPen\WObj:=wPaper;
    MoveL Offs(pOrigin,251.70,162.89,0.00),v40,z0,tPen\WObj:=wPaper;
    MoveL Offs(pOrigin,250.85,162.04,0.00),v40,fine,tPen\WObj:=wPaper;
    MoveL Offs(pOrigin,250.85,162.04,6.00),v60,z5,tPen\WObj:=wPaper;
    MoveL Offs(pOrigin,251.91,162.84,6.00),vTravel,z5,tPen\WObj:=wPaper;
    MoveL Offs(pOrigin,251.91,162.84,0.00),v60,z0,tPen\WObj:=wPaper;
    MoveL Offs(pOrigin,253.19,162.84,0.00),v40,z0,tPen\WObj:=wPaper;
    MoveL Offs(pOrigin,253.82,163.10,0.00),v40,z0,tPen\WObj:=wPaper;
    MoveL Offs(pOrigin,254.25,163.52,0.00),v40,z0,tPen\WObj:=wPaper;
    MoveL Offs(pOrigin,253.82,163.10,0.00),v40,z0,tPen\WObj:=wPaper;
    MoveL Offs(pOrigin,254.25,163.90,0.00),v40,z0,tPen\WObj:=wPaper;
    MoveL Offs(pOrigin,251.91,163.90,0.00),v40,z0,tPen\WObj:=wPaper;
    MoveL Offs(pOrigin,251.27,164.38,0.00),v40,z0,tPen\WObj:=wPaper;
    MoveL Offs(pOrigin,250.64,165.01,0.00),v40,z0,tPen\WObj:=wPaper;
    MoveL Offs(pOrigin,251.27,164.38,0.00),v40,z0,tPen\WObj:=wPaper;
    MoveL Offs(pOrigin,251.06,164.95,0.00),v40,z0,tPen\WObj:=wPaper;
    MoveL Offs(pOrigin,252.55,164.95,0.00),v40,z0,tPen\WObj:=wPaper;
    MoveL Offs(pOrigin,252.34,165.01,0.00),v40,z0,tPen\WObj:=wPaper;
    MoveL Offs(pOrigin,252.12,165.44,0.00),v40,z0,tPen\WObj:=wPaper;
    MoveL Offs(pOrigin,252.34,165.01,0.00),v40,z0,tPen\WObj:=wPaper;
    MoveL Offs(pOrigin,252.13,165.81,0.00),v40,z0,tPen\WObj:=wPaper;
    MoveL Offs(pOrigin,250.63,164.30,0.00),v40,fine,tPen\WObj:=wPaper;
    MoveL Offs(pOrigin,250.63,164.30,6.00),v60,z5,tPen\WObj:=wPaper;
    MoveL Offs(pOrigin,248.94,163.10,6.00),vTravel,z5,tPen\WObj:=wPaper;
    MoveL Offs(pOrigin,248.94,163.10,0.00),v60,z0,tPen\WObj:=wPaper;
    MoveL Offs(pOrigin,248.09,163.24,0.00),v40,z0,tPen\WObj:=wPaper;
    MoveL Offs(pOrigin,242.14,167.07,0.00),v40,z0,tPen\WObj:=wPaper;
  ENDPROC

  PROC DrawPart172()
    MoveL Offs(pOrigin,241.29,167.35,0.00),v40,z0,tPen\WObj:=wPaper;
    MoveL Offs(pOrigin,240.93,167.14,0.00),v40,z0,tPen\WObj:=wPaper;
    MoveL Offs(pOrigin,241.22,165.86,0.00),v40,z0,tPen\WObj:=wPaper;
    MoveL Offs(pOrigin,244.12,161.61,0.00),v40,z0,tPen\WObj:=wPaper;
    MoveL Offs(pOrigin,246.18,157.79,0.00),v40,z0,tPen\WObj:=wPaper;
    MoveL Offs(pOrigin,246.82,158.14,0.00),v40,z0,tPen\WObj:=wPaper;
    MoveL Offs(pOrigin,248.92,156.04,0.00),v40,z0,tPen\WObj:=wPaper;
    MoveL Offs(pOrigin,249.52,156.94,0.00),v40,z0,tPen\WObj:=wPaper;
    MoveL Offs(pOrigin,247.41,159.04,0.00),v40,z0,tPen\WObj:=wPaper;
    MoveL Offs(pOrigin,248.01,159.94,0.00),v40,z0,tPen\WObj:=wPaper;
    MoveL Offs(pOrigin,249.96,157.99,0.00),v40,z0,tPen\WObj:=wPaper;
    MoveL Offs(pOrigin,249.15,158.00,0.00),v40,z0,tPen\WObj:=wPaper;
    MoveL Offs(pOrigin,249.79,158.85,0.00),v40,z0,tPen\WObj:=wPaper;
    MoveL Offs(pOrigin,249.15,158.00,0.00),v40,fine,tPen\WObj:=wPaper;
    MoveL Offs(pOrigin,249.15,158.00,6.00),v60,z5,tPen\WObj:=wPaper;
    MoveL Offs(pOrigin,250.86,158.58,6.00),vTravel,z5,tPen\WObj:=wPaper;
    MoveL Offs(pOrigin,250.86,158.58,0.00),v60,z0,tPen\WObj:=wPaper;
    MoveL Offs(pOrigin,248.61,160.84,0.00),v40,z0,tPen\WObj:=wPaper;
    MoveL Offs(pOrigin,249.57,160.55,0.00),v40,z0,tPen\WObj:=wPaper;
    MoveL Offs(pOrigin,250.00,160.98,0.00),v40,z0,tPen\WObj:=wPaper;
    MoveL Offs(pOrigin,249.57,160.55,0.00),v40,z0,tPen\WObj:=wPaper;
    MoveL Offs(pOrigin,249.35,161.58,0.00),v40,z0,tPen\WObj:=wPaper;
    MoveL Offs(pOrigin,251.46,159.48,0.00),v40,fine,tPen\WObj:=wPaper;
    MoveL Offs(pOrigin,251.46,159.48,6.00),v60,z5,tPen\WObj:=wPaper;
    MoveL Offs(pOrigin,252.66,156.78,6.00),vTravel,z5,tPen\WObj:=wPaper;
    MoveL Offs(pOrigin,252.66,156.78,0.00),v60,z0,tPen\WObj:=wPaper;
    MoveL Offs(pOrigin,257.02,152.42,0.00),v40,z0,tPen\WObj:=wPaper;
    MoveL Offs(pOrigin,256.16,152.48,0.00),v40,z0,tPen\WObj:=wPaper;
    MoveL Offs(pOrigin,255.81,151.41,0.00),v40,z0,tPen\WObj:=wPaper;
    MoveL Offs(pOrigin,254.89,150.35,0.00),v40,z0,tPen\WObj:=wPaper;
    MoveL Offs(pOrigin,252.98,149.93,0.00),v40,z0,tPen\WObj:=wPaper;
    MoveL Offs(pOrigin,251.20,150.99,0.00),v40,z0,tPen\WObj:=wPaper;
    MoveL Offs(pOrigin,250.64,152.05,0.00),v40,z0,tPen\WObj:=wPaper;
    MoveL Offs(pOrigin,250.64,153.54,0.00),v40,z0,tPen\WObj:=wPaper;
    MoveL Offs(pOrigin,251.27,154.81,0.00),v40,z0,tPen\WObj:=wPaper;
    MoveL Offs(pOrigin,251.91,155.31,0.00),v40,z0,tPen\WObj:=wPaper;
    MoveL Offs(pOrigin,254.04,155.66,0.00),v40,z0,tPen\WObj:=wPaper;
    MoveL Offs(pOrigin,255.60,154.60,0.00),v40,z0,tPen\WObj:=wPaper;
    MoveL Offs(pOrigin,256.16,153.32,0.00),v40,z0,tPen\WObj:=wPaper;
    MoveL Offs(pOrigin,256.16,152.48,0.00),v40,z0,tPen\WObj:=wPaper;
    MoveL Offs(pOrigin,255.98,151.74,0.00),v40,z0,tPen\WObj:=wPaper;
    MoveL Offs(pOrigin,254.18,149.93,0.00),v40,z0,tPen\WObj:=wPaper;
    MoveL Offs(pOrigin,254.49,148.98,0.00),v40,z0,tPen\WObj:=wPaper;
    MoveL Offs(pOrigin,249.68,153.79,0.00),v40,z0,tPen\WObj:=wPaper;
    MoveL Offs(pOrigin,250.60,153.82,0.00),v40,z0,tPen\WObj:=wPaper;
    MoveL Offs(pOrigin,252.55,155.77,0.00),v40,z0,tPen\WObj:=wPaper;
    MoveL Offs(pOrigin,251.62,156.33,0.00),v40,z0,tPen\WObj:=wPaper;
    MoveL Offs(pOrigin,256.73,151.22,0.00),v40,z0,tPen\WObj:=wPaper;
    MoveL Offs(pOrigin,256.13,150.33,0.00),v40,z0,tPen\WObj:=wPaper;
    MoveL Offs(pOrigin,250.72,155.74,0.00),v40,z0,tPen\WObj:=wPaper;
    MoveL Offs(pOrigin,250.12,154.84,0.00),v40,z0,tPen\WObj:=wPaper;
    MoveL Offs(pOrigin,255.38,149.58,0.00),v40,fine,tPen\WObj:=wPaper;
    MoveL Offs(pOrigin,255.38,149.58,6.00),v60,z5,tPen\WObj:=wPaper;
    MoveL Offs(pOrigin,252.99,148.99,6.00),vTravel,z5,tPen\WObj:=wPaper;
    MoveL Offs(pOrigin,252.99,148.99,0.00),v60,z0,tPen\WObj:=wPaper;
    MoveL Offs(pOrigin,249.53,152.44,0.00),v40,fine,tPen\WObj:=wPaper;
    MoveL Offs(pOrigin,249.53,152.44,6.00),v60,z5,tPen\WObj:=wPaper;
    MoveL Offs(pOrigin,252.76,153.54,6.00),vTravel,z5,tPen\WObj:=wPaper;
    MoveL Offs(pOrigin,252.76,153.54,0.00),v60,z0,tPen\WObj:=wPaper;
    MoveL Offs(pOrigin,253.61,153.54,0.00),v40,z0,tPen\WObj:=wPaper;
    MoveL Offs(pOrigin,254.04,153.11,0.00),v40,z0,tPen\WObj:=wPaper;
    MoveL Offs(pOrigin,253.82,152.48,0.00),v40,z0,tPen\WObj:=wPaper;
    MoveL Offs(pOrigin,252.98,152.26,0.00),v40,fine,tPen\WObj:=wPaper;
    MoveL Offs(pOrigin,252.98,152.26,6.00),v60,z5,tPen\WObj:=wPaper;
    MoveL Offs(pOrigin,257.02,153.92,6.00),vTravel,z5,tPen\WObj:=wPaper;
    MoveL Offs(pOrigin,257.02,153.92,0.00),v60,z0,tPen\WObj:=wPaper;
    MoveL Offs(pOrigin,254.46,156.47,0.00),v40,fine,tPen\WObj:=wPaper;
    MoveL Offs(pOrigin,254.46,156.47,6.00),v60,z5,tPen\WObj:=wPaper;
    MoveL Offs(pOrigin,253.61,164.80,6.00),vTravel,z5,tPen\WObj:=wPaper;
    MoveL Offs(pOrigin,253.61,164.80,0.00),v60,z0,tPen\WObj:=wPaper;
    MoveL Offs(pOrigin,254.04,165.23,0.00),v40,z0,tPen\WObj:=wPaper;
    MoveL Offs(pOrigin,253.61,164.80,0.00),v40,z0,tPen\WObj:=wPaper;
    MoveL Offs(pOrigin,254.04,164.95,0.00),v40,z0,tPen\WObj:=wPaper;
    MoveL Offs(pOrigin,255.52,164.95,0.00),v40,z0,tPen\WObj:=wPaper;
    MoveL Offs(pOrigin,256.68,164.71,0.00),v40,z0,tPen\WObj:=wPaper;
    MoveL Offs(pOrigin,254.58,166.81,0.00),v40,fine,tPen\WObj:=wPaper;
    MoveL Offs(pOrigin,254.58,166.81,6.00),v60,z5,tPen\WObj:=wPaper;
    MoveL Offs(pOrigin,254.25,165.44,6.00),vTravel,z5,tPen\WObj:=wPaper;
    MoveL Offs(pOrigin,254.25,165.44,0.00),v60,z0,tPen\WObj:=wPaper;
    MoveL Offs(pOrigin,254.68,165.86,0.00),v40,z0,tPen\WObj:=wPaper;
    MoveL Offs(pOrigin,254.25,165.44,0.00),v40,fine,tPen\WObj:=wPaper;
    MoveL Offs(pOrigin,254.25,165.44,6.00),v60,z5,tPen\WObj:=wPaper;
    MoveL Offs(pOrigin,256.59,165.65,6.00),vTravel,z5,tPen\WObj:=wPaper;
    MoveL Offs(pOrigin,256.59,165.65,0.00),v60,z0,tPen\WObj:=wPaper;
    MoveL Offs(pOrigin,257.01,166.07,0.00),v40,z0,tPen\WObj:=wPaper;
    MoveL Offs(pOrigin,256.59,165.65,0.00),v40,fine,tPen\WObj:=wPaper;
    MoveL Offs(pOrigin,256.59,165.65,6.00),v60,z5,tPen\WObj:=wPaper;
    MoveL Offs(pOrigin,258.71,170.11,6.00),vTravel,z5,tPen\WObj:=wPaper;
    MoveL Offs(pOrigin,258.71,170.11,0.00),v60,z0,tPen\WObj:=wPaper;
    MoveL Offs(pOrigin,258.92,170.54,0.00),v40,z0,tPen\WObj:=wPaper;
    MoveL Offs(pOrigin,258.71,170.11,0.00),v40,z0,tPen\WObj:=wPaper;
    MoveL Offs(pOrigin,258.92,170.23,0.00),v40,z0,tPen\WObj:=wPaper;
    MoveL Offs(pOrigin,259.99,170.23,0.00),v40,z0,tPen\WObj:=wPaper;
    MoveL Offs(pOrigin,260.41,171.29,0.00),v40,z0,tPen\WObj:=wPaper;
    MoveL Offs(pOrigin,259.35,171.29,0.00),v40,fine,tPen\WObj:=wPaper;
    MoveL Offs(pOrigin,259.35,171.29,6.00),v60,z5,tPen\WObj:=wPaper;
    MoveL Offs(pOrigin,258.31,172.04,6.00),vTravel,z5,tPen\WObj:=wPaper;
    MoveL Offs(pOrigin,258.31,172.04,0.00),v60,z0,tPen\WObj:=wPaper;
    MoveL Offs(pOrigin,260.86,169.49,0.00),v40,fine,tPen\WObj:=wPaper;
    MoveL Offs(pOrigin,260.86,169.49,6.00),v60,z5,tPen\WObj:=wPaper;
    MoveL Offs(pOrigin,261.16,170.68,6.00),vTravel,z5,tPen\WObj:=wPaper;
    MoveL Offs(pOrigin,261.16,170.68,0.00),v60,z0,tPen\WObj:=wPaper;
    MoveL Offs(pOrigin,258.61,173.24,0.00),v40,z0,tPen\WObj:=wPaper;
    MoveL Offs(pOrigin,259.04,172.72,0.00),v40,z0,tPen\WObj:=wPaper;
    MoveL Offs(pOrigin,262.65,176.32,0.00),v40,z0,tPen\WObj:=wPaper;
    MoveL Offs(pOrigin,262.33,176.27,0.00),v40,z0,tPen\WObj:=wPaper;
    MoveL Offs(pOrigin,262.75,176.91,0.00),v40,z0,tPen\WObj:=wPaper;
    MoveL Offs(pOrigin,262.33,176.27,0.00),v40,z0,tPen\WObj:=wPaper;
    MoveL Offs(pOrigin,262.32,176.57,0.00),v40,z0,tPen\WObj:=wPaper;
    MoveL Offs(pOrigin,261.05,176.57,0.00),v40,z0,tPen\WObj:=wPaper;
    MoveL Offs(pOrigin,261.48,177.62,0.00),v40,z0,tPen\WObj:=wPaper;
    MoveL Offs(pOrigin,263.18,177.62,0.00),v40,z0,tPen\WObj:=wPaper;
    MoveL Offs(pOrigin,263.60,178.19,0.00),v40,z0,tPen\WObj:=wPaper;
    MoveL Offs(pOrigin,263.81,178.61,0.00),v40,z0,tPen\WObj:=wPaper;
    MoveL Offs(pOrigin,263.60,178.19,0.00),v40,z0,tPen\WObj:=wPaper;
    MoveL Offs(pOrigin,263.81,178.68,0.00),v40,z0,tPen\WObj:=wPaper;
    MoveL Offs(pOrigin,262.11,178.68,0.00),v40,z0,tPen\WObj:=wPaper;
    MoveL Offs(pOrigin,261.43,179.37,0.00),v40,z0,tPen\WObj:=wPaper;
    MoveL Offs(pOrigin,263.69,177.12,0.00),v40,z0,tPen\WObj:=wPaper;
    MoveL Offs(pOrigin,264.28,178.01,0.00),v40,z0,tPen\WObj:=wPaper;
  ENDPROC

  PROC DrawPart173()
    MoveL Offs(pOrigin,262.03,180.27,0.00),v40,z0,tPen\WObj:=wPaper;
    MoveL Offs(pOrigin,262.96,179.89,0.00),v40,z0,tPen\WObj:=wPaper;
    MoveL Offs(pOrigin,263.39,180.31,0.00),v40,z0,tPen\WObj:=wPaper;
    MoveL Offs(pOrigin,262.96,179.89,0.00),v40,z0,tPen\WObj:=wPaper;
    MoveL Offs(pOrigin,263.18,179.74,0.00),v40,z0,tPen\WObj:=wPaper;
    MoveL Offs(pOrigin,264.45,179.74,0.00),v40,z0,tPen\WObj:=wPaper;
    MoveL Offs(pOrigin,264.66,179.89,0.00),v40,z0,tPen\WObj:=wPaper;
    MoveL Offs(pOrigin,265.09,180.31,0.00),v40,z0,tPen\WObj:=wPaper;
    MoveL Offs(pOrigin,264.66,179.89,0.00),v40,z0,tPen\WObj:=wPaper;
    MoveL Offs(pOrigin,265.30,180.79,0.00),v40,z0,tPen\WObj:=wPaper;
    MoveL Offs(pOrigin,264.02,180.79,0.00),v40,fine,tPen\WObj:=wPaper;
    MoveL Offs(pOrigin,264.02,180.79,6.00),v60,z5,tPen\WObj:=wPaper;
    MoveL Offs(pOrigin,262.78,181.02,6.00),vTravel,z5,tPen\WObj:=wPaper;
    MoveL Offs(pOrigin,262.78,181.02,0.00),v60,z0,tPen\WObj:=wPaper;
    MoveL Offs(pOrigin,265.18,178.61,0.00),v40,fine,tPen\WObj:=wPaper;
    MoveL Offs(pOrigin,265.18,178.61,6.00),v60,z5,tPen\WObj:=wPaper;
    MoveL Offs(pOrigin,265.94,177.34,6.00),vTravel,z5,tPen\WObj:=wPaper;
    MoveL Offs(pOrigin,265.94,177.34,0.00),v60,z0,tPen\WObj:=wPaper;
    MoveL Offs(pOrigin,271.60,186.48,0.00),v40,z0,tPen\WObj:=wPaper;
    MoveL Offs(pOrigin,272.95,187.96,0.00),v40,z0,tPen\WObj:=wPaper;
    MoveL Offs(pOrigin,272.95,187.96,0.00),v40,z0,tPen\WObj:=wPaper;
    MoveL Offs(pOrigin,272.10,187.32,0.00),v40,fine,tPen\WObj:=wPaper;
    MoveL Offs(pOrigin,272.10,187.32,6.00),v60,z5,tPen\WObj:=wPaper;
    MoveL Offs(pOrigin,272.80,185.93,6.00),vTravel,z5,tPen\WObj:=wPaper;
    MoveL Offs(pOrigin,272.80,185.93,0.00),v60,z0,tPen\WObj:=wPaper;
    MoveL Offs(pOrigin,268.44,190.29,0.00),v40,z0,tPen\WObj:=wPaper;
    MoveL Offs(pOrigin,269.19,191.03,0.00),v40,z0,tPen\WObj:=wPaper;
    MoveL Offs(pOrigin,273.54,186.67,0.00),v40,z0,tPen\WObj:=wPaper;
    MoveL Offs(pOrigin,273.77,187.44,0.00),v40,z0,tPen\WObj:=wPaper;
    MoveL Offs(pOrigin,275.57,189.25,0.00),v40,z0,tPen\WObj:=wPaper;
    MoveL Offs(pOrigin,274.88,189.82,0.00),v40,z0,tPen\WObj:=wPaper;
    MoveL Offs(pOrigin,278.64,186.06,0.00),v40,z0,tPen\WObj:=wPaper;
    MoveL Offs(pOrigin,278.11,185.81,0.00),v40,z0,tPen\WObj:=wPaper;
    MoveL Offs(pOrigin,276.45,184.16,0.00),v40,z0,tPen\WObj:=wPaper;
    MoveL Offs(pOrigin,275.80,184.42,0.00),v40,z0,tPen\WObj:=wPaper;
    MoveL Offs(pOrigin,282.86,177.36,0.00),v40,z0,tPen\WObj:=wPaper;
    MoveL Offs(pOrigin,281.88,177.62,0.00),v40,z0,tPen\WObj:=wPaper;
    MoveL Offs(pOrigin,278.26,177.62,0.00),v40,z0,tPen\WObj:=wPaper;
    MoveL Offs(pOrigin,278.05,178.68,0.00),v40,z0,tPen\WObj:=wPaper;
    MoveL Offs(pOrigin,279.32,178.68,0.00),v40,fine,tPen\WObj:=wPaper;
    MoveL Offs(pOrigin,279.32,178.68,6.00),v60,z5,tPen\WObj:=wPaper;
    MoveL Offs(pOrigin,281.02,178.68,6.00),vTravel,z5,tPen\WObj:=wPaper;
    MoveL Offs(pOrigin,281.02,178.68,0.00),v60,z0,tPen\WObj:=wPaper;
    MoveL Offs(pOrigin,282.09,178.68,0.00),v40,z0,tPen\WObj:=wPaper;
    MoveL Offs(pOrigin,282.30,179.74,0.00),v40,z0,tPen\WObj:=wPaper;
    MoveL Offs(pOrigin,281.24,179.74,0.00),v40,z0,tPen\WObj:=wPaper;
    MoveL Offs(pOrigin,281.66,180.79,0.00),v40,z0,tPen\WObj:=wPaper;
    MoveL Offs(pOrigin,282.73,180.79,0.00),v40,z0,tPen\WObj:=wPaper;
    MoveL Offs(pOrigin,283.75,180.95,0.00),v40,z0,tPen\WObj:=wPaper;
    MoveL Offs(pOrigin,281.04,183.66,0.00),v40,fine,tPen\WObj:=wPaper;
    MoveL Offs(pOrigin,281.04,183.66,6.00),v60,z5,tPen\WObj:=wPaper;
    MoveL Offs(pOrigin,282.09,182.90,6.00),vTravel,z5,tPen\WObj:=wPaper;
    MoveL Offs(pOrigin,282.09,182.90,0.00),v60,z0,tPen\WObj:=wPaper;
    MoveL Offs(pOrigin,283.15,182.90,0.00),v40,z0,tPen\WObj:=wPaper;
    MoveL Offs(pOrigin,283.36,183.96,0.00),v40,z0,tPen\WObj:=wPaper;
    MoveL Offs(pOrigin,282.30,183.96,0.00),v40,z0,tPen\WObj:=wPaper;
    MoveL Offs(pOrigin,282.51,185.02,0.00),v40,z0,tPen\WObj:=wPaper;
    MoveL Offs(pOrigin,283.79,185.02,0.00),v40,z0,tPen\WObj:=wPaper;
    MoveL Offs(pOrigin,284.25,184.48,0.00),v40,z0,tPen\WObj:=wPaper;
    MoveL Offs(pOrigin,280.94,181.17,0.00),v40,z0,tPen\WObj:=wPaper;
    MoveL Offs(pOrigin,281.88,181.85,0.00),v40,z0,tPen\WObj:=wPaper;
    MoveL Offs(pOrigin,282.94,181.85,0.00),v40,fine,tPen\WObj:=wPaper;
    MoveL Offs(pOrigin,282.94,181.85,6.00),v60,z5,tPen\WObj:=wPaper;
    MoveL Offs(pOrigin,284.34,183.35,6.00),vTravel,z5,tPen\WObj:=wPaper;
    MoveL Offs(pOrigin,284.34,183.35,0.00),v60,z0,tPen\WObj:=wPaper;
    MoveL Offs(pOrigin,281.64,186.05,0.00),v40,fine,tPen\WObj:=wPaper;
    MoveL Offs(pOrigin,281.64,186.05,6.00),v60,z5,tPen\WObj:=wPaper;
    MoveL Offs(pOrigin,281.93,187.25,6.00),vTravel,z5,tPen\WObj:=wPaper;
    MoveL Offs(pOrigin,281.93,187.25,0.00),v60,z0,tPen\WObj:=wPaper;
    MoveL Offs(pOrigin,284.64,184.54,0.00),v40,fine,tPen\WObj:=wPaper;
    MoveL Offs(pOrigin,284.64,184.54,6.00),v60,z5,tPen\WObj:=wPaper;
    MoveL Offs(pOrigin,284.00,186.07,6.00),vTravel,z5,tPen\WObj:=wPaper;
    MoveL Offs(pOrigin,284.00,186.07,0.00),v60,z0,tPen\WObj:=wPaper;
    MoveL Offs(pOrigin,282.94,186.07,0.00),v40,z0,tPen\WObj:=wPaper;
    MoveL Offs(pOrigin,283.15,187.13,0.00),v40,z0,tPen\WObj:=wPaper;
    MoveL Offs(pOrigin,284.21,187.13,0.00),v40,z0,tPen\WObj:=wPaper;
    MoveL Offs(pOrigin,285.23,186.94,0.00),v40,z0,tPen\WObj:=wPaper;
    MoveL Offs(pOrigin,282.67,189.49,0.00),v40,z0,tPen\WObj:=wPaper;
    MoveL Offs(pOrigin,283.58,189.24,0.00),v40,z0,tPen\WObj:=wPaper;
    MoveL Offs(pOrigin,284.85,189.24,0.00),v40,z0,tPen\WObj:=wPaper;
    MoveL Offs(pOrigin,285.82,189.33,0.00),v40,z0,tPen\WObj:=wPaper;
    MoveL Offs(pOrigin,283.27,191.89,0.00),v40,z0,tPen\WObj:=wPaper;
    MoveL Offs(pOrigin,284.21,191.35,0.00),v40,z0,tPen\WObj:=wPaper;
    MoveL Offs(pOrigin,285.27,191.35,0.00),v40,z0,tPen\WObj:=wPaper;
    MoveL Offs(pOrigin,285.76,190.48,0.00),v40,z0,tPen\WObj:=wPaper;
    MoveL Offs(pOrigin,282.46,187.17,0.00),v40,fine,tPen\WObj:=wPaper;
    MoveL Offs(pOrigin,282.46,187.17,6.00),v60,z5,tPen\WObj:=wPaper;
    MoveL Offs(pOrigin,283.36,188.18,6.00),vTravel,z5,tPen\WObj:=wPaper;
    MoveL Offs(pOrigin,283.36,188.18,0.00),v60,z0,tPen\WObj:=wPaper;
    MoveL Offs(pOrigin,284.42,188.18,0.00),v40,fine,tPen\WObj:=wPaper;
    MoveL Offs(pOrigin,284.42,188.18,6.00),v60,z5,tPen\WObj:=wPaper;
    MoveL Offs(pOrigin,283.79,190.30,6.00),vTravel,z5,tPen\WObj:=wPaper;
    MoveL Offs(pOrigin,283.79,190.30,0.00),v60,z0,tPen\WObj:=wPaper;
    MoveL Offs(pOrigin,285.06,190.30,0.00),v40,z0,tPen\WObj:=wPaper;
    MoveL Offs(pOrigin,286.12,190.53,0.00),v40,z0,tPen\WObj:=wPaper;
    MoveL Offs(pOrigin,283.41,193.24,0.00),v40,z0,tPen\WObj:=wPaper;
    MoveL Offs(pOrigin,283.82,193.02,0.00),v40,z0,tPen\WObj:=wPaper;
    MoveL Offs(pOrigin,287.13,196.32,0.00),v40,z0,tPen\WObj:=wPaper;
    MoveL Offs(pOrigin,287.75,196.37,0.00),v40,z0,tPen\WObj:=wPaper;
    MoveL Offs(pOrigin,284.89,199.22,0.00),v40,z0,tPen\WObj:=wPaper;
    MoveL Offs(pOrigin,285.34,200.27,0.00),v40,z0,tPen\WObj:=wPaper;
    MoveL Offs(pOrigin,293.60,192.01,0.00),v40,z0,tPen\WObj:=wPaper;
    MoveL Offs(pOrigin,294.16,192.90,0.00),v40,z0,tPen\WObj:=wPaper;
    MoveL Offs(pOrigin,295.06,193.80,0.00),v40,z0,tPen\WObj:=wPaper;
    MoveL Offs(pOrigin,295.26,192.85,0.00),v40,z0,tPen\WObj:=wPaper;
    MoveL Offs(pOrigin,296.33,192.64,0.00),v40,z0,tPen\WObj:=wPaper;
    MoveL Offs(pOrigin,296.54,192.00,0.00),v40,z0,tPen\WObj:=wPaper;
    MoveL Offs(pOrigin,296.54,192.00,0.00),v40,z0,tPen\WObj:=wPaper;
    MoveL Offs(pOrigin,297.39,191.79,0.00),v40,z0,tPen\WObj:=wPaper;
    MoveL Offs(pOrigin,297.39,191.36,0.00),v40,z0,tPen\WObj:=wPaper;
    MoveL Offs(pOrigin,297.17,190.94,0.00),v40,z0,tPen\WObj:=wPaper;
    MoveL Offs(pOrigin,296.54,191.15,0.00),v40,z0,tPen\WObj:=wPaper;
    MoveL Offs(pOrigin,296.33,191.79,0.00),v40,z0,tPen\WObj:=wPaper;
    MoveL Offs(pOrigin,296.33,191.79,0.00),v40,z0,tPen\WObj:=wPaper;
    MoveL Offs(pOrigin,295.69,191.79,0.00),v40,z0,tPen\WObj:=wPaper;
    MoveL Offs(pOrigin,295.26,192.21,0.00),v40,z0,tPen\WObj:=wPaper;
    MoveL Offs(pOrigin,295.26,192.85,0.00),v40,z0,tPen\WObj:=wPaper;
    MoveL Offs(pOrigin,295.26,192.85,0.00),v40,z0,tPen\WObj:=wPaper;
    MoveL Offs(pOrigin,294.41,193.27,0.00),v40,z0,tPen\WObj:=wPaper;
    MoveL Offs(pOrigin,293.56,194.34,0.00),v40,z0,tPen\WObj:=wPaper;
  ENDPROC

  PROC DrawPart174()
    MoveL Offs(pOrigin,293.77,194.12,0.00),v40,z0,tPen\WObj:=wPaper;
    MoveL Offs(pOrigin,294.16,194.40,0.00),v40,z0,tPen\WObj:=wPaper;
    MoveL Offs(pOrigin,293.26,193.50,0.00),v40,fine,tPen\WObj:=wPaper;
    MoveL Offs(pOrigin,293.26,193.50,6.00),v60,z5,tPen\WObj:=wPaper;
    MoveL Offs(pOrigin,294.75,192.00,6.00),vTravel,z5,tPen\WObj:=wPaper;
    MoveL Offs(pOrigin,294.75,192.00,0.00),v60,z0,tPen\WObj:=wPaper;
    MoveL Offs(pOrigin,295.96,193.20,0.00),v40,z0,tPen\WObj:=wPaper;
    MoveL Offs(pOrigin,296.70,192.46,0.00),v40,z0,tPen\WObj:=wPaper;
    MoveL Offs(pOrigin,295.65,191.41,0.00),v40,z0,tPen\WObj:=wPaper;
    MoveL Offs(pOrigin,296.55,190.81,0.00),v40,z0,tPen\WObj:=wPaper;
    MoveL Offs(pOrigin,297.60,191.86,0.00),v40,z0,tPen\WObj:=wPaper;
    MoveL Offs(pOrigin,297.95,192.14,0.00),v40,z0,tPen\WObj:=wPaper;
    MoveL Offs(pOrigin,304.86,185.23,0.00),v40,fine,tPen\WObj:=wPaper;
    MoveL Offs(pOrigin,304.86,185.23,6.00),v60,z5,tPen\WObj:=wPaper;
    MoveL Offs(pOrigin,304.02,186.34,6.00),vTravel,z5,tPen\WObj:=wPaper;
    MoveL Offs(pOrigin,304.02,186.34,0.00),v60,z0,tPen\WObj:=wPaper;
    MoveL Offs(pOrigin,305.68,187.99,0.00),v40,fine,tPen\WObj:=wPaper;
    MoveL Offs(pOrigin,305.68,187.99,6.00),v60,z5,tPen\WObj:=wPaper;
    MoveL Offs(pOrigin,304.40,188.18,6.00),vTravel,z5,tPen\WObj:=wPaper;
    MoveL Offs(pOrigin,304.40,188.18,0.00),v60,z0,tPen\WObj:=wPaper;
    MoveL Offs(pOrigin,301.00,188.18,0.00),v40,z0,tPen\WObj:=wPaper;
    MoveL Offs(pOrigin,301.03,187.83,0.00),v40,z0,tPen\WObj:=wPaper;
    MoveL Offs(pOrigin,304.04,190.83,0.00),v40,z0,tPen\WObj:=wPaper;
    MoveL Offs(pOrigin,303.98,190.30,0.00),v40,z0,tPen\WObj:=wPaper;
    MoveL Offs(pOrigin,304.40,190.51,0.00),v40,z0,tPen\WObj:=wPaper;
    MoveL Offs(pOrigin,303.98,190.30,0.00),v40,z0,tPen\WObj:=wPaper;
    MoveL Offs(pOrigin,304.61,190.30,0.00),v40,z0,tPen\WObj:=wPaper;
    MoveL Offs(pOrigin,306.95,190.30,0.00),v40,z0,tPen\WObj:=wPaper;
    MoveL Offs(pOrigin,306.79,189.27,0.00),v40,z0,tPen\WObj:=wPaper;
    MoveL Offs(pOrigin,304.69,191.37,0.00),v40,fine,tPen\WObj:=wPaper;
    MoveL Offs(pOrigin,304.69,191.37,6.00),v60,z5,tPen\WObj:=wPaper;
    MoveL Offs(pOrigin,305.25,189.24,6.00),vTravel,z5,tPen\WObj:=wPaper;
    MoveL Offs(pOrigin,305.25,189.24,0.00),v60,z0,tPen\WObj:=wPaper;
    MoveL Offs(pOrigin,302.49,189.24,0.00),v40,z0,tPen\WObj:=wPaper;
    MoveL Offs(pOrigin,303.09,189.02,0.00),v40,z0,tPen\WObj:=wPaper;
    MoveL Offs(pOrigin,303.09,187.75,0.00),v40,fine,tPen\WObj:=wPaper;
    MoveL Offs(pOrigin,303.09,187.75,6.00),v60,z5,tPen\WObj:=wPaper;
    MoveL Offs(pOrigin,300.58,189.66,6.00),vTravel,z5,tPen\WObj:=wPaper;
    MoveL Offs(pOrigin,300.58,189.66,0.00),v60,z0,tPen\WObj:=wPaper;
    MoveL Offs(pOrigin,301.00,189.45,0.00),v40,z0,tPen\WObj:=wPaper;
    MoveL Offs(pOrigin,300.58,189.66,0.00),v40,z0,tPen\WObj:=wPaper;
    MoveL Offs(pOrigin,300.29,190.07,0.00),v40,z0,tPen\WObj:=wPaper;
    MoveL Offs(pOrigin,299.24,189.02,0.00),v40,z0,tPen\WObj:=wPaper;
    MoveL Offs(pOrigin,298.19,189.47,0.00),v40,z0,tPen\WObj:=wPaper;
    MoveL Offs(pOrigin,299.24,190.52,0.00),v40,z0,tPen\WObj:=wPaper;
    MoveL Offs(pOrigin,298.50,191.26,0.00),v40,z0,tPen\WObj:=wPaper;
    MoveL Offs(pOrigin,297.30,190.06,0.00),v40,fine,tPen\WObj:=wPaper;
    MoveL Offs(pOrigin,297.30,190.06,6.00),v60,z5,tPen\WObj:=wPaper;
    MoveL Offs(pOrigin,306.63,192.41,6.00),vTravel,z5,tPen\WObj:=wPaper;
    MoveL Offs(pOrigin,306.63,192.41,0.00),v60,z0,tPen\WObj:=wPaper;
    MoveL Offs(pOrigin,308.89,190.16,0.00),v40,z0,tPen\WObj:=wPaper;
    MoveL Offs(pOrigin,309.93,190.61,0.00),v40,z0,tPen\WObj:=wPaper;
    MoveL Offs(pOrigin,307.68,192.86,0.00),v40,z0,tPen\WObj:=wPaper;
    MoveL Offs(pOrigin,307.59,192.00,0.00),v40,z0,tPen\WObj:=wPaper;
    MoveL Offs(pOrigin,308.01,192.21,0.00),v40,z0,tPen\WObj:=wPaper;
    MoveL Offs(pOrigin,307.59,192.00,0.00),v40,z0,tPen\WObj:=wPaper;
    MoveL Offs(pOrigin,306.95,191.35,0.00),v40,z0,tPen\WObj:=wPaper;
    MoveL Offs(pOrigin,309.08,191.35,0.00),v40,z0,tPen\WObj:=wPaper;
    MoveL Offs(pOrigin,310.14,191.79,0.00),v40,z0,tPen\WObj:=wPaper;
    MoveL Offs(pOrigin,310.56,192.00,0.00),v40,z0,tPen\WObj:=wPaper;
    MoveL Offs(pOrigin,310.14,191.79,0.00),v40,fine,tPen\WObj:=wPaper;
    MoveL Offs(pOrigin,310.14,191.79,6.00),v60,z5,tPen\WObj:=wPaper;
    MoveL Offs(pOrigin,310.35,193.27,6.00),vTravel,z5,tPen\WObj:=wPaper;
    MoveL Offs(pOrigin,310.35,193.27,0.00),v60,z0,tPen\WObj:=wPaper;
    MoveL Offs(pOrigin,310.77,193.49,0.00),v40,z0,tPen\WObj:=wPaper;
    MoveL Offs(pOrigin,310.35,193.27,0.00),v40,fine,tPen\WObj:=wPaper;
    MoveL Offs(pOrigin,310.35,193.27,6.00),v60,z5,tPen\WObj:=wPaper;
    MoveL Offs(pOrigin,311.40,198.20,6.00),vTravel,z5,tPen\WObj:=wPaper;
    MoveL Offs(pOrigin,311.40,198.20,0.00),v60,z0,tPen\WObj:=wPaper;
    MoveL Offs(pOrigin,312.75,199.55,0.00),v40,z0,tPen\WObj:=wPaper;
    MoveL Offs(pOrigin,311.84,200.29,0.00),v40,z0,tPen\WObj:=wPaper;
    MoveL Offs(pOrigin,311.20,200.93,0.00),v40,z0,tPen\WObj:=wPaper;
    MoveL Offs(pOrigin,311.84,200.29,0.00),v40,fine,tPen\WObj:=wPaper;
    MoveL Offs(pOrigin,311.84,200.29,6.00),v60,z5,tPen\WObj:=wPaper;
    MoveL Offs(pOrigin,311.55,202.44,6.00),vTravel,z5,tPen\WObj:=wPaper;
    MoveL Offs(pOrigin,311.55,202.44,0.00),v60,z0,tPen\WObj:=wPaper;
    MoveL Offs(pOrigin,286.90,227.08,0.00),v40,z0,tPen\WObj:=wPaper;
    MoveL Offs(pOrigin,287.40,226.20,0.00),v40,z0,tPen\WObj:=wPaper;
    MoveL Offs(pOrigin,289.52,226.20,0.00),v40,z0,tPen\WObj:=wPaper;
    MoveL Offs(pOrigin,289.52,226.21,0.00),v40,z0,tPen\WObj:=wPaper;
    MoveL Offs(pOrigin,289.74,225.79,0.00),v40,z0,tPen\WObj:=wPaper;
    MoveL Offs(pOrigin,289.52,226.21,0.00),v40,z0,tPen\WObj:=wPaper;
    MoveL Offs(pOrigin,290.07,226.14,0.00),v40,z0,tPen\WObj:=wPaper;
    MoveL Offs(pOrigin,281.95,218.03,0.00),v40,z0,tPen\WObj:=wPaper;
    MoveL Offs(pOrigin,281.24,217.81,0.00),v40,z0,tPen\WObj:=wPaper;
    MoveL Offs(pOrigin,282.59,216.46,0.00),v40,z0,tPen\WObj:=wPaper;
    MoveL Offs(pOrigin,281.84,215.71,0.00),v40,z0,tPen\WObj:=wPaper;
    MoveL Offs(pOrigin,280.64,216.91,0.00),v40,z0,tPen\WObj:=wPaper;
    MoveL Offs(pOrigin,280.20,215.86,0.00),v40,z0,tPen\WObj:=wPaper;
    MoveL Offs(pOrigin,281.10,214.96,0.00),v40,fine,tPen\WObj:=wPaper;
    MoveL Offs(pOrigin,281.10,214.96,6.00),v60,z5,tPen\WObj:=wPaper;
    MoveL Offs(pOrigin,282.45,213.61,6.00),vTravel,z5,tPen\WObj:=wPaper;
    MoveL Offs(pOrigin,282.45,213.61,0.00),v60,z0,tPen\WObj:=wPaper;
    MoveL Offs(pOrigin,284.70,211.36,0.00),v40,z0,tPen\WObj:=wPaper;
    MoveL Offs(pOrigin,284.18,211.29,0.00),v40,z0,tPen\WObj:=wPaper;
    MoveL Offs(pOrigin,274.71,201.83,0.00),v40,fine,tPen\WObj:=wPaper;
    MoveL Offs(pOrigin,274.71,201.83,6.00),v60,z5,tPen\WObj:=wPaper;
    MoveL Offs(pOrigin,273.64,203.00,6.00),vTravel,z5,tPen\WObj:=wPaper;
    MoveL Offs(pOrigin,273.64,203.00,0.00),v60,z0,tPen\WObj:=wPaper;
    MoveL Offs(pOrigin,278.00,198.64,0.00),v40,z0,tPen\WObj:=wPaper;
    MoveL Offs(pOrigin,277.55,198.69,0.00),v40,z0,tPen\WObj:=wPaper;
    MoveL Offs(pOrigin,265.98,187.12,0.00),v40,z0,tPen\WObj:=wPaper;
    MoveL Offs(pOrigin,266.05,188.20,0.00),v40,z0,tPen\WObj:=wPaper;
    MoveL Offs(pOrigin,270.86,183.39,0.00),v40,z0,tPen\WObj:=wPaper;
    MoveL Offs(pOrigin,270.26,182.49,0.00),v40,z0,tPen\WObj:=wPaper;
    MoveL Offs(pOrigin,265.00,187.75,0.00),v40,z0,tPen\WObj:=wPaper;
    MoveL Offs(pOrigin,264.11,187.15,0.00),v40,z0,tPen\WObj:=wPaper;
    MoveL Offs(pOrigin,269.67,181.59,0.00),v40,z0,tPen\WObj:=wPaper;
    MoveL Offs(pOrigin,269.07,180.70,0.00),v40,z0,tPen\WObj:=wPaper;
    MoveL Offs(pOrigin,265.16,184.60,0.00),v40,z0,tPen\WObj:=wPaper;
    MoveL Offs(pOrigin,264.41,185.35,0.00),v40,z0,tPen\WObj:=wPaper;
    MoveL Offs(pOrigin,263.06,186.71,0.00),v40,z0,tPen\WObj:=wPaper;
    MoveL Offs(pOrigin,262.01,186.26,0.00),v40,z0,tPen\WObj:=wPaper;
    MoveL Offs(pOrigin,263.21,185.06,0.00),v40,fine,tPen\WObj:=wPaper;
    MoveL Offs(pOrigin,263.21,185.06,6.00),v60,z5,tPen\WObj:=wPaper;
    MoveL Offs(pOrigin,262.02,184.76,6.00),vTravel,z5,tPen\WObj:=wPaper;
    MoveL Offs(pOrigin,262.02,184.76,0.00),v60,z0,tPen\WObj:=wPaper;
    MoveL Offs(pOrigin,260.96,185.81,0.00),v40,fine,tPen\WObj:=wPaper;
    MoveL Offs(pOrigin,260.96,185.81,6.00),v60,z5,tPen\WObj:=wPaper;
    MoveL Offs(pOrigin,259.14,184.77,6.00),vTravel,z5,tPen\WObj:=wPaper;
  ENDPROC

  PROC DrawPart175()
    MoveL Offs(pOrigin,259.14,184.77,0.00),v60,z0,tPen\WObj:=wPaper;
    MoveL Offs(pOrigin,263.17,185.98,0.00),v40,z0,tPen\WObj:=wPaper;
    MoveL Offs(pOrigin,268.27,188.18,0.00),v40,z0,tPen\WObj:=wPaper;
    MoveL Offs(pOrigin,268.27,188.18,0.00),v40,z0,tPen\WObj:=wPaper;
    MoveL Offs(pOrigin,269.34,189.88,0.00),v40,z0,tPen\WObj:=wPaper;
    MoveL Offs(pOrigin,271.04,191.57,0.00),v40,z0,tPen\WObj:=wPaper;
    MoveL Offs(pOrigin,273.73,195.61,0.00),v40,z0,tPen\WObj:=wPaper;
    MoveL Offs(pOrigin,273.80,196.68,0.00),v40,z0,tPen\WObj:=wPaper;
    MoveL Offs(pOrigin,273.38,196.63,0.00),v40,z0,tPen\WObj:=wPaper;
    MoveL Offs(pOrigin,275.92,196.63,0.00),v40,z0,tPen\WObj:=wPaper;
    MoveL Offs(pOrigin,275.71,196.25,0.00),v40,z0,tPen\WObj:=wPaper;
    MoveL Offs(pOrigin,276.14,196.89,0.00),v40,z0,tPen\WObj:=wPaper;
    MoveL Offs(pOrigin,275.71,196.25,0.00),v40,z0,tPen\WObj:=wPaper;
    MoveL Offs(pOrigin,276.36,195.80,0.00),v40,z0,tPen\WObj:=wPaper;
    MoveL Offs(pOrigin,273.66,198.51,0.00),v40,z0,tPen\WObj:=wPaper;
    MoveL Offs(pOrigin,274.23,197.69,0.00),v40,z0,tPen\WObj:=wPaper;
    MoveL Offs(pOrigin,276.56,197.69,0.00),v40,z0,tPen\WObj:=wPaper;
    MoveL Offs(pOrigin,277.56,197.60,0.00),v40,z0,tPen\WObj:=wPaper;
    MoveL Offs(pOrigin,272.90,202.26,0.00),v40,z0,tPen\WObj:=wPaper;
    MoveL Offs(pOrigin,272.00,201.66,0.00),v40,z0,tPen\WObj:=wPaper;
    MoveL Offs(pOrigin,273.35,200.31,0.00),v40,fine,tPen\WObj:=wPaper;
    MoveL Offs(pOrigin,273.35,200.31,6.00),v60,z5,tPen\WObj:=wPaper;
    MoveL Offs(pOrigin,274.25,199.41,6.00),vTravel,z5,tPen\WObj:=wPaper;
    MoveL Offs(pOrigin,274.25,199.41,0.00),v60,z0,tPen\WObj:=wPaper;
    MoveL Offs(pOrigin,276.96,196.70,0.00),v40,fine,tPen\WObj:=wPaper;
    MoveL Offs(pOrigin,276.96,196.70,6.00),v60,z5,tPen\WObj:=wPaper;
    MoveL Offs(pOrigin,275.63,197.31,6.00),vTravel,z5,tPen\WObj:=wPaper;
    MoveL Offs(pOrigin,275.63,197.31,0.00),v60,z0,tPen\WObj:=wPaper;
    MoveL Offs(pOrigin,275.63,198.80,0.00),v40,z0,tPen\WObj:=wPaper;
    MoveL Offs(pOrigin,275.29,198.80,0.00),v40,z0,tPen\WObj:=wPaper;
    MoveL Offs(pOrigin,276.14,199.65,0.00),v40,z0,tPen\WObj:=wPaper;
    MoveL Offs(pOrigin,275.29,198.80,0.00),v40,z0,tPen\WObj:=wPaper;
    MoveL Offs(pOrigin,275.08,198.74,0.00),v40,z0,tPen\WObj:=wPaper;
    MoveL Offs(pOrigin,277.20,198.74,0.00),v40,z0,tPen\WObj:=wPaper;
    MoveL Offs(pOrigin,277.41,199.01,0.00),v40,z0,tPen\WObj:=wPaper;
    MoveL Offs(pOrigin,277.62,199.44,0.00),v40,z0,tPen\WObj:=wPaper;
    MoveL Offs(pOrigin,277.41,199.01,0.00),v40,z0,tPen\WObj:=wPaper;
    MoveL Offs(pOrigin,277.84,199.65,0.00),v40,z0,tPen\WObj:=wPaper;
    MoveL Offs(pOrigin,278.05,200.07,0.00),v40,z0,tPen\WObj:=wPaper;
    MoveL Offs(pOrigin,277.84,199.65,0.00),v40,z0,tPen\WObj:=wPaper;
    MoveL Offs(pOrigin,277.62,199.80,0.00),v40,z0,tPen\WObj:=wPaper;
    MoveL Offs(pOrigin,276.14,199.80,0.00),v40,fine,tPen\WObj:=wPaper;
    MoveL Offs(pOrigin,276.14,199.80,6.00),v60,z5,tPen\WObj:=wPaper;
    MoveL Offs(pOrigin,278.60,199.54,6.00),vTravel,z5,tPen\WObj:=wPaper;
    MoveL Offs(pOrigin,278.60,199.54,0.00),v60,z0,tPen\WObj:=wPaper;
    MoveL Offs(pOrigin,274.54,203.60,0.00),v40,fine,tPen\WObj:=wPaper;
    MoveL Offs(pOrigin,274.54,203.60,6.00),v60,z5,tPen\WObj:=wPaper;
    MoveL Offs(pOrigin,276.03,205.09,6.00),vTravel,z5,tPen\WObj:=wPaper;
    MoveL Offs(pOrigin,276.03,205.09,0.00),v60,z0,tPen\WObj:=wPaper;
    MoveL Offs(pOrigin,279.64,201.49,0.00),v40,z0,tPen\WObj:=wPaper;
    MoveL Offs(pOrigin,280.24,202.38,0.00),v40,z0,tPen\WObj:=wPaper;
    MoveL Offs(pOrigin,276.93,205.69,0.00),v40,z0,tPen\WObj:=wPaper;
    MoveL Offs(pOrigin,277.53,206.59,0.00),v40,z0,tPen\WObj:=wPaper;
    MoveL Offs(pOrigin,280.68,203.43,0.00),v40,z0,tPen\WObj:=wPaper;
    MoveL Offs(pOrigin,280.18,204.02,0.00),v40,z0,tPen\WObj:=wPaper;
    MoveL Offs(pOrigin,278.26,204.02,0.00),v40,z0,tPen\WObj:=wPaper;
    MoveL Offs(pOrigin,278.48,204.96,0.00),v40,z0,tPen\WObj:=wPaper;
    MoveL Offs(pOrigin,278.48,203.90,0.00),v40,z0,tPen\WObj:=wPaper;
    MoveL Offs(pOrigin,277.91,202.62,0.00),v40,z0,tPen\WObj:=wPaper;
    MoveL Offs(pOrigin,273.80,196.89,0.00),v40,z0,tPen\WObj:=wPaper;
    MoveL Offs(pOrigin,265.73,192.57,0.00),v40,z0,tPen\WObj:=wPaper;
    MoveL Offs(pOrigin,259.56,190.94,0.00),v40,z0,tPen\WObj:=wPaper;
    MoveL Offs(pOrigin,257.01,190.94,0.00),v40,z0,tPen\WObj:=wPaper;
    MoveL Offs(pOrigin,251.06,192.21,0.00),v40,z0,tPen\WObj:=wPaper;
    MoveL Offs(pOrigin,246.18,191.15,0.00),v40,z0,tPen\WObj:=wPaper;
    MoveL Offs(pOrigin,243.62,190.94,0.00),v40,z0,tPen\WObj:=wPaper;
    MoveL Offs(pOrigin,238.31,192.35,0.00),v40,z0,tPen\WObj:=wPaper;
    MoveL Offs(pOrigin,233.21,194.98,0.00),v40,z0,tPen\WObj:=wPaper;
    MoveL Offs(pOrigin,232.36,196.68,0.00),v40,z0,tPen\WObj:=wPaper;
    MoveL Offs(pOrigin,230.24,199.01,0.00),v40,z0,tPen\WObj:=wPaper;
    MoveL Offs(pOrigin,228.40,201.77,0.00),v40,z0,tPen\WObj:=wPaper;
    MoveL Offs(pOrigin,228.54,202.34,0.00),v40,z0,tPen\WObj:=wPaper;
    MoveL Offs(pOrigin,229.39,202.62,0.00),v40,z0,tPen\WObj:=wPaper;
    MoveL Offs(pOrigin,229.39,202.62,0.00),v40,z0,tPen\WObj:=wPaper;
    MoveL Offs(pOrigin,233.21,200.22,0.00),v40,z0,tPen\WObj:=wPaper;
    MoveL Offs(pOrigin,236.40,198.73,0.00),v40,z0,tPen\WObj:=wPaper;
    MoveL Offs(pOrigin,240.44,197.38,0.00),v40,z0,tPen\WObj:=wPaper;
    MoveL Offs(pOrigin,240.86,197.52,0.00),v40,z0,tPen\WObj:=wPaper;
    MoveL Offs(pOrigin,240.41,197.41,0.00),v40,z0,tPen\WObj:=wPaper;
    MoveL Offs(pOrigin,239.50,198.31,0.00),v40,fine,tPen\WObj:=wPaper;
    MoveL Offs(pOrigin,239.50,198.31,6.00),v60,z5,tPen\WObj:=wPaper;
    MoveL Offs(pOrigin,243.41,198.16,6.00),vTravel,z5,tPen\WObj:=wPaper;
    MoveL Offs(pOrigin,243.41,198.16,0.00),v60,z0,tPen\WObj:=wPaper;
    MoveL Offs(pOrigin,248.09,200.29,0.00),v40,z0,tPen\WObj:=wPaper;
    MoveL Offs(pOrigin,248.09,200.29,0.00),v40,z0,tPen\WObj:=wPaper;
    MoveL Offs(pOrigin,248.30,201.14,0.00),v40,z0,tPen\WObj:=wPaper;
    MoveL Offs(pOrigin,249.79,200.93,0.00),v40,z0,tPen\WObj:=wPaper;
    MoveL Offs(pOrigin,249.79,200.93,0.00),v40,z0,tPen\WObj:=wPaper;
    MoveL Offs(pOrigin,249.36,200.29,0.00),v40,z0,tPen\WObj:=wPaper;
    MoveL Offs(pOrigin,248.09,200.29,0.00),v40,z0,tPen\WObj:=wPaper;
    MoveL Offs(pOrigin,248.79,199.48,0.00),v40,z0,tPen\WObj:=wPaper;
    MoveL Offs(pOrigin,247.14,201.14,0.00),v40,z0,tPen\WObj:=wPaper;
    MoveL Offs(pOrigin,246.39,200.39,0.00),v40,z0,tPen\WObj:=wPaper;
    MoveL Offs(pOrigin,247.59,199.19,0.00),v40,z0,tPen\WObj:=wPaper;
    MoveL Offs(pOrigin,246.54,198.74,0.00),v40,z0,tPen\WObj:=wPaper;
    MoveL Offs(pOrigin,245.34,199.94,0.00),v40,z0,tPen\WObj:=wPaper;
    MoveL Offs(pOrigin,244.75,199.05,0.00),v40,z0,tPen\WObj:=wPaper;
    MoveL Offs(pOrigin,245.65,198.14,0.00),v40,fine,tPen\WObj:=wPaper;
    MoveL Offs(pOrigin,245.65,198.14,6.00),v60,z5,tPen\WObj:=wPaper;
    MoveL Offs(pOrigin,248.18,201.58,6.00),vTravel,z5,tPen\WObj:=wPaper;
    MoveL Offs(pOrigin,248.18,201.58,0.00),v60,z0,tPen\WObj:=wPaper;
    MoveL Offs(pOrigin,249.99,199.78,0.00),v40,z0,tPen\WObj:=wPaper;
    MoveL Offs(pOrigin,249.39,200.40,0.00),v40,z0,tPen\WObj:=wPaper;
    MoveL Offs(pOrigin,250.14,201.15,0.00),v40,z0,tPen\WObj:=wPaper;
    MoveL Offs(pOrigin,249.79,200.93,0.00),v40,z0,tPen\WObj:=wPaper;
    MoveL Offs(pOrigin,252.98,201.14,0.00),v40,z0,tPen\WObj:=wPaper;
    MoveL Offs(pOrigin,257.01,200.50,0.00),v40,z0,tPen\WObj:=wPaper;
    MoveL Offs(pOrigin,259.99,200.50,0.00),v40,z0,tPen\WObj:=wPaper;
    MoveL Offs(pOrigin,265.09,201.99,0.00),v40,fine,tPen\WObj:=wPaper;
    MoveL Offs(pOrigin,265.09,201.99,6.00),v60,z5,tPen\WObj:=wPaper;
    MoveL Offs(pOrigin,262.57,200.64,6.00),vTravel,z5,tPen\WObj:=wPaper;
    MoveL Offs(pOrigin,262.57,200.64,0.00),v60,z0,tPen\WObj:=wPaper;
    MoveL Offs(pOrigin,261.67,201.54,0.00),v40,fine,tPen\WObj:=wPaper;
    MoveL Offs(pOrigin,261.67,201.54,6.00),v60,z5,tPen\WObj:=wPaper;
    MoveL Offs(pOrigin,260.32,201.40,6.00),vTravel,z5,tPen\WObj:=wPaper;
    MoveL Offs(pOrigin,260.32,201.40,0.00),v60,z0,tPen\WObj:=wPaper;
    MoveL Offs(pOrigin,261.67,200.04,0.00),v40,fine,tPen\WObj:=wPaper;
    MoveL Offs(pOrigin,261.67,200.04,6.00),v60,z5,tPen\WObj:=wPaper;
    MoveL Offs(pOrigin,260.47,199.75,6.00),vTravel,z5,tPen\WObj:=wPaper;
    MoveL Offs(pOrigin,260.47,199.75,0.00),v60,z0,tPen\WObj:=wPaper;
  ENDPROC

